# B&R Automation Studio project BottlePlant2
Automation Studio 4.10.2.37; technology packages: Acp10Arnc0 5.12.2, mapp 5.12.1, mappSafety 5.12.2

## Configuration Config1

CPU 4PPC70.0702-20W, AutomationRuntime B4.91, Build 4.1.2, Safety 0.0, Vc V4.72.3

### Task classes (Cpu.sw)
```
Cyclic#1 (cycle 2000 us):
  AxisCtrl <- Software.Code.AxisCtrl.prg
  RobVis <- Source.Misc.RobVis.prg
  MachineSta <- Software.Code.MachineCtrl.prg
DataObjects: Acp10sys
NcDataObjects: acp10etxen <- acp10etxen.dob, gTranAxisa <- gTranAxisobj.gTranAxisa.dob, gTranAxisi <- gTranAxisobj.gTranAxisi.dob, gCartAxisa <- gCartAxisobj.gCartAxisa.dob, gCartAxisi <- gCartAxisobj.gCartAxisi.dob, gPourAxisa <- gPourAxisobj.gPourAxisa.dob, gPourAxisi <- gPourAxisobj.gPourAxisi.dob
VcDataObjects: Visu <- Software.HMI.Visu.dob
Binaries: udbdef, arflatprv, TCData, arsvcreg, FWRules, arcoal, acp10cfg, Acp10map, sysconf, iomap, asfw, Transport, Role, ashwac, Cart, Pourer, arconfig, ashwd, User
Libraries: SfDomain, Acp10man, Acp10par, NcGlobal, Acp10sim, Acp10_MC, sys_lib, brsystem, runtime, MpAxis, MpBase, MpCom, astcp, asieccon, fileio, asbrstr, asiodiag, SfDomVis, astime, dataobj, SfDomDrv, asusb, MpSfDomMgr, aruser, powerlnk, standard, AsBrMath
```

### Task classes (AppMo.sw)
```

```

### Hardware
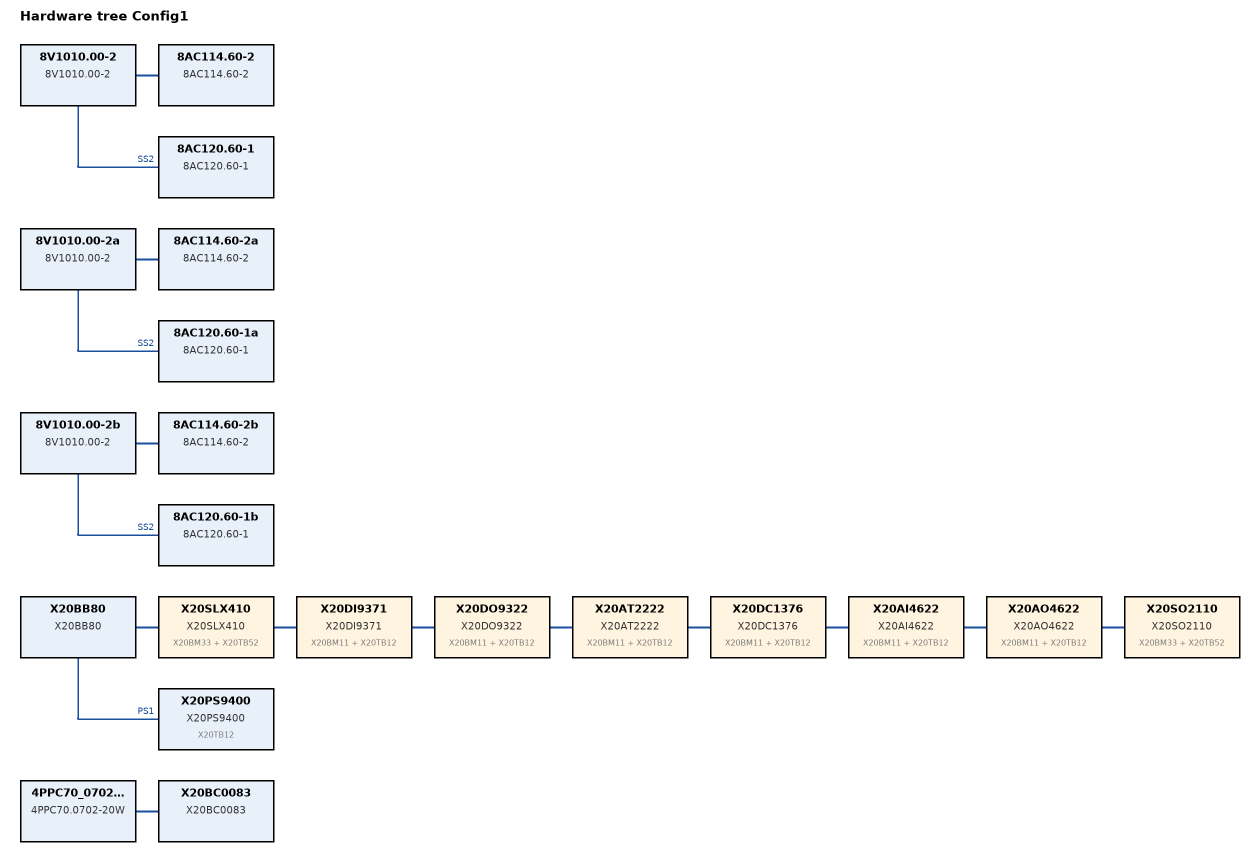
```
4PPC70_0702_20W : 4PPC70.0702-20W v1.5.2.0
  Connector IF2:
    ActivateDevice = 1
    Mode = Manual
    InternetAddress = 10.48.30.236
    SubnetMask = 255.255.255.0
    Vnc1
    VncVcObjectName1 = Visu
    VncKeyMappingFile1 = VC\PS2-Keyboard.dis
    VncRefreshRate1 = 100
    ActivateSnmp = 2
  ConfigurationID = BottlePlant2_Config1
  Simulation = 1
  TimerDeviceType = EPLX2X
  TimerDevice = 4PPC70_0702_20W.IF1
  TaskClassIdleTime = 2000
  Cyclic1Duration = 2000
  FileDevice1
  FileDeviceName1 = RecipeFile
  FileDevicePath1 = F:\Recipe
  FtpUser1
  FtpUsername1 = Admin
  FtpUserPassword1 = uT8p0uNS80JC7A4YbQtDpgpyP3aiMc7PVyx0K6ICeRY=
  FtpUserSalt1 = sviO6ryF
  FTPAccessRight1 = 0
  ActivateOpcUa = 1
  OpcUaInformationModels_PV_Version = 1
  VcObjectName = Visu
  KeyMappingFile = VC\4PPC70_0702_20W.dis
8AC114.60-2 : 8AC114.60-2 v1.0.0.8  [SS -> 8V1010.00-2.SS1; PLK1 -> X20BC0083.PLK2 (NodeNumber=4) [Cable Type=PowerlinkCable, Length=10, Version=1.0.0.3]; PLK2 -> 8AC114.60-2a.PLK1 (NodeNumber=4) [Cable Type=PowerlinkCable, Length=10, Version=1.0.0.3]]
8AC114.60-2a : 8AC114.60-2 v1.0.0.8  [SS -> 8V1010.00-2a.SS1; PLK1 -> 8AC114.60-2.PLK2 (NodeNumber=6) [Cable Type=PowerlinkCable, Length=10, Version=1.0.0.3]; PLK2 -> 8AC114.60-2b.PLK1 (NodeNumber=6) [Cable Type=PowerlinkCable, Length=10, Version=1.0.0.3]]
8AC114.60-2b : 8AC114.60-2 v1.0.0.8  [SS -> 8V1010.00-2b.SS1; PLK1 -> 8AC114.60-2a.PLK2 (NodeNumber=9) [Cable Type=PowerlinkCable, Length=10, Version=1.0.0.3]]
8AC120.60-1 : 8AC120.60-1 v2.2.0.0  [SS -> 8V1010.00-2.SS2]
8AC120.60-1a : 8AC120.60-1 v2.2.0.0  [SS -> 8V1010.00-2a.SS2]
8AC120.60-1b : 8AC120.60-1 v2.2.0.0  [SS -> 8V1010.00-2b.SS2]
8V1010.00-2 : 8V1010.00-2 v2.2.0.0
  MotionTP = Acp10Arnc0
  Simulate = standard
  PoweredBy = DC
  ActiveMotorSimulation_r1 = on
  BothEndSwitchesAreNormallyOpen_r1 = on
  QuickStopIsNormallyOpen_r1 = on
8V1010.00-2a : 8V1010.00-2 v2.2.0.0
  MotionTP = Acp10Arnc0
  Simulate = standard
  PoweredBy = DC
  ActiveMotorSimulation_r1 = on
  BothEndSwitchesAreNormallyOpen_r1 = on
  QuickStopIsNormallyOpen_r1 = on
8V1010.00-2b : 8V1010.00-2 v2.2.0.0
  MotionTP = Acp10Arnc0
  Simulate = standard
  PoweredBy = DC
  ActiveMotorSimulation_r1 = on
  BothEndSwitchesAreNormallyOpen_r1 = on
  QuickStopIsNormallyOpen_r1 = on
X20AI4622 : X20AI4622 v1.1.0.0  [SS1 -> X20TB12e.SS; SL -> X20BM11d.SL1]
  Supervision = off
X20AO4622 : X20AO4622 v1.2.0.0  [SS1 -> X20TB12f.SS; SL -> X20BM11e.SL1]
  Supervision = off
X20AT2222 : X20AT2222 v1.3.0.0  [SS1 -> X20TB12c.SS; SL -> X20BM11b.SL1]
  Supervision = off
X20BB80 : X20BB80 v1.0.2.0
X20BC0083 : X20BC0083 v2.11.1.0  [PLK1 -> 4PPC70_0702_20W.IF1 (NodeNumber=2) [Cable Type=PowerlinkCable, Length=10, Version=1.0.0.3]; PLK2 -> 8AC114.60-2.PLK1 (NodeNumber=2) [Cable Type=PowerlinkCable, Length=10, Version=1.0.0.3]; SL -> X20BB80.SL1]
  Supervision = off
X20BM11 : X20BM11 v1.0.0.1  [X2X1 -> X20BM33.X2X2]
X20BM11a : X20BM11 v1.0.0.1  [X2X1 -> X20BM11.X2X2]
X20BM11b : X20BM11 v1.0.0.1  [X2X1 -> X20BM11a.X2X2]
X20BM11c : X20BM11 v1.0.0.1  [X2X1 -> X20BM11b.X2X2]
X20BM11d : X20BM11 v1.0.0.1  [X2X1 -> X20BM11c.X2X2]
X20BM11e : X20BM11 v1.0.0.1  [X2X1 -> X20BM11d.X2X2]
X20BM33 : X20BM33 v1.0.0.6  [X2X1 -> X20BB80.IF1]
X20BM33a : X20BM33 v1.0.0.6  [X2X1 -> X20BM11e.X2X2]
X20DC1376 : X20DC1376 v1.2.0.0  [SS1 -> X20TB12d.SS; SL -> X20BM11c.SL1]
  Supervision = off
X20DI9371 : X20DI9371 v1.1.0.0  [SS1 -> X20TB12a.SS; SL -> X20BM11.SL1]
  Supervision = off
X20DO9322 : X20DO9322 v1.3.0.0  [SS1 -> X20TB12b.SS; SL -> X20BM11a.SL1]
  Supervision = off
X20PS9400 : X20PS9400 v1.5.0.0  [SS1 -> X20TB12.SS; PS -> X20BB80.PS1]
  Supervision = off
X20SLX410 : X20SLX410 v2.4.0.1  [SS1 -> X20TB52.SS; SL -> X20BM33.SL1]
  Supervision = off
X20SO2110 : X20SO2110 v2.2.1.0  [SS1 -> X20TB52a.SS; SL -> X20BM33a.SL1]
  Supervision = off
X20TB12 : X20TB12 v1.0.0.0
X20TB12a : X20TB12 v1.0.0.0
X20TB12b : X20TB12 v1.0.0.0
X20TB12c : X20TB12 v1.0.0.0
X20TB12d : X20TB12 v1.0.0.0
X20TB12e : X20TB12 v1.0.0.0
X20TB12f : X20TB12 v1.0.0.0
X20TB52 : X20TB52 v1.0.0.2
X20TB52a : X20TB52 v1.0.0.2
```

### IoMap.iom - 4PPC70_0702_20W/IoMap.iom
```iecst
VAR_CONFIG
	::SequencerC:DoPourer AT %QX."X20DO9322".DigitalOutput01;
END_VAR
```

### Acp10cfg.ncc - 4PPC70_0702_20W/Motion/Acp10cfg.ncc
```
NcConfiguration (Version=5.12.2, NcSwId=Acp10)
  ACP10CF1_typ:
    cnt_nettrc_rec_drive = 1500
    bufsize_trace_upload = 1200
    tc_nc_man_task = Cyclic #1
    glob_pv_as_ncobject = Yes
    ncsys_dl_broadcast = Yes
    ncsys_dl_acp_reset = Yes
    safemc_log_err_to_ax = Yes
    network_init:
      ncsw_init_execute = Yes
      automatic_execute = No
      node_nr_warning = Yes
      net_err_before_ncact = Yes
    nettrc:
      enter_parsecrec = Yes
      enter_ncaction = Yes
      save_ring_startidx = Yes
    cam_prof_download:
      cam_dat_dl_parallel = No
      tc_cam_dl_parallel = Task class for NC Manager task
    plk_if[0]:
      if_name = IF1
      tc_CycDat_PLCopen = Task class for NC Manager task
      mc_broadcast_extdat = No
```

### Acp10map.ncm - 4PPC70_0702_20W/Motion/Acp10map.ncm
```
NcMapping (NcSwId=Acp10, DisabledNodesAreHidden=False)
  NcObject gTranAxis (ModuleId=8V1010.00-2, Type=ncAXIS, Channel=1, AcoposSimulation=Standard, InitParameter=gTranAxisi, AcoposParameter=gTranAxisa, Disabled=FALSE, ModuleDisabled=FALSE)
  NcObject 8V1010.00-2_ncV_AXIS1 (ModuleId=8V1010.00-2, Type=ncV_AXIS, Channel=1, Disabled=TRUE, ModuleDisabled=FALSE)
  NcObject gCartAxis (ModuleId=8V1010.00-2a, Type=ncAXIS, Channel=1, AcoposSimulation=Standard, InitParameter=gCartAxisi, AcoposParameter=gCartAxisa, Disabled=FALSE, ModuleDisabled=FALSE)
  NcObject 8V1010.00-2a_ncV_AXIS1 (ModuleId=8V1010.00-2a, Type=ncV_AXIS, Channel=1, Disabled=TRUE, ModuleDisabled=FALSE)
  NcObject gPourAxis (ModuleId=8V1010.00-2b, Type=ncAXIS, Channel=1, AcoposSimulation=Standard, InitParameter=gPourAxisi, AcoposParameter=gPourAxisa, Disabled=FALSE, ModuleDisabled=FALSE)
  NcObject 8V1010.00-2b_ncV_AXIS1 (ModuleId=8V1010.00-2b, Type=ncV_AXIS, Channel=1, Disabled=TRUE, ModuleDisabled=FALSE)
```

### Cart.mpaxisbasic - 4PPC70_0702_20W/Motion/Config/Cart.mpaxisbasic
```
Element gCartAxisCfg (Type=mpaxisbasic)
  AxisConfiguration = AxisWithConfiguration
    Axis:
      BaseType = 4
    Drive:
      Controller:
        LoopFilters:
          [0]
          [1]
          [2]
Element gCartAxisCfg_1 (Type=mpaxisbasic)
```

### Pourer.mpaxisbasic - 4PPC70_0702_20W/Motion/Config/Pourer.mpaxisbasic
```
Element gPourAxisCfg (Type=mpaxisbasic)
  AxisConfiguration = AxisWithConfiguration
    Axis:
      BaseType = 4
      PeriodSettings:
        Period = 360
      MovementLimits:
        VelocityPositive = 1000
        VelocityNegative = 1000
        Acceleration = 5000
        Deceleration = 5000
    Drive:
      Controller:
        LoopFilters:
          [0]
          [1]
          [2]
```

### Transport.mpaxisbasic - 4PPC70_0702_20W/Motion/Config/Transport.mpaxisbasic
```
Element gTranAxisCfg (Type=mpaxisbasic)
  AxisConfiguration = AxisWithConfiguration
    Axis:
      BaseType = 4
      PeriodSettings:
        Period = 360
    Drive:
      Controller:
        LoopFilters:
          [0]
          [1]
          [2]
```

### Alarm.mpalarmbasic - 4PPC70_0702_20W/mappServices/Alarm/Alarm.mpalarmbasic
```
Element gAlarmBasic (Type=mpalarmbasic)
  mapp.Alarm.Factory:
    Reactions:
      Reaction[0]:
        Description = Example: Immediate Stop
  Alarms:
    UserAlarm:
      Alarms:
        Alarm[0]:
          Description = Example: Temperature over Tolerance
          Reaction = 1
```

### UserManagm.mpuser - 4PPC70_0702_20W/mappServices/User/UserManagm.mpuser
```
Element UserMgmt (Type=mpuser)
  Groups:
    DefGroup#1:
      id = Admin
      level = 100
      admin = TRUE
      rights:
        [0] = FullAccess
        [1] = FullAccess
        [2] = FullAccess
        [3] = FullAccess
        [4] = FullAccess
    DefGroup#2:
      id = Operator
      rights:
        [0] = FullAccess
        [1] = StartOnly
        [2] = ViewOnly
        [3] = ViewOnly
        [4] = NoAccess
    DefGroup#3:
      id = Supervisor
      level = 21
  Users:
    DefUser#1:
      id = Admin
      grp = Admin
      name = Default Admin User
      pwd = Admin
      pref = /LANG=0 /UNIT=0
    DefUser#2:
      id = macko
      grp = Operator
      pwd = 12345
    DefUser#3:
      id = supervisor1
      grp = Supervisor
      pwd = 12345
```

### UserSign.mpusersign - 4PPC70_0702_20W/mappServices/User/UserSign.mpusersign
```
Element gUserSign (Type=mpusersign)
```

## Logical view

Binary libraries used (declarations not repeated): operator, runtime, astime, AsIecCon, SfDomain 5.12.2, Acp10man, Acp10par, NcGlobal, Acp10sim, Acp10_MC, sys_lib, brsystem, MpAxis, MpBase, MpCom, standard, AsBrMath, MpRecipe, asstring, FileIO, MpUser 5.12.1, MpFile, MpAlarm 5.12.1

### Global.typ - Global data types
```iecst
(* AutoAxis *)
TYPE
	gAxesCtrlType : 	STRUCT
		Ctrl : gAxisBasicCtrlType;
		Cmd : gCmdType;
		State : gAutoAxisStateType;
		Timers : gTimersType;
		TimersPar : gTimersParType;
	END_STRUCT;
	gAxisBasicCtrlType : 	STRUCT
		MpTransporterAxis : MpAxisBasic;
		MpTransporterAxisPar : MpAxisBasicParType;
		MpCartAxis : MpAxisBasic;
		MpCartAxisPar : MpAxisBasicParType;
		MpPourerAxis : MpAxisBasic;
		MpPourerAxisPar : MpAxisBasicParType;
	END_STRUCT;
	gCmdType : 	STRUCT
		Power : BOOL;
		Home : BOOL;
		Update : BOOL;
		Stop : BOOL;
		ErrorReset : BOOL;
		MoveVelocity : BOOL;
		MoveAdditive : BOOL;
		MoveAbsolute : BOOL;
	END_STRUCT;

	gTimersType : STRUCT
		PowerTimer : ARRAY[0..2] OF TON;
		HomeTimer : ARRAY[0..2] OF TON;
	END_STRUCT;

	gTimersParType : STRUCT
		PowerDelayTime : REAL :=5;
		HomeDelayTime : REAL :=5;
	END_STRUCT;

	gAutoAxisStateType :
		(
		STATE_INIT_AXES := 0,
		STATE_WAIT_FOR_CMD_AXES := 1,
		STATE_POWER_ON_AXES := 2,
		STATE_HOME_AXES := 3,
		STATE_UPDATE_AXES := 4,
		STATE_MOVE_VELOCITY_AXES := 5,
		STATE_MOVE_ABSOLUTE_AXES := 6,
		STATE_MOVE_ADDITIVE_AXES := 7,
		STATE_STOP_AXES := 8,
		STATE_ERROR_AXES := 10
	);
END_TYPE
```

### Global.var - Global variables
```iecst
VAR
	gTranAxis : ACP10AXIS_typ;
	gCartAxis : ACP10AXIS_typ;
	gPourAxis : ACP10AXIS_typ;
END_VAR
```


### Program Logical/Software/Code/AxisCtrl (IEC)

#### Main.st
```iecst
PROGRAM _INIT
	(* Insert code here *)
	gAxes.SequencerCtrl.MpAxisCamSequencer_0.Enable:=TRUE;
	gAxes.SequencerCtrl.MpAxisCamSequencer_1.Enable:=TRUE;

	gAxes.SequencerCtrl.MpAxisCamSequencerPar_0.Deceleration:=1000;
	gAxes.SequencerCtrl.MpAxisCamSequencerPar_0.Configuration.Master:=ADR(gTranAxis);
	gAxes.SequencerCtrl.MpAxisCamSequencerPar_0.Configuration.StartState:=0;
	gAxes.SequencerCtrl.MpAxisCamSequencerPar_0.Configuration.State[0].Event[0].Type:=ncS_START;
	gAxes.SequencerCtrl.MpAxisCamSequencerPar_0.Configuration.State[0].Event[0].Attribute:=ncAT_ONCE;
	gAxes.SequencerCtrl.MpAxisCamSequencerPar_0.Configuration.State[0].Event[0].NextState:=1;

	gAxes.SequencerCtrl.MpAxisCamSequencerPar_0.Configuration.State[1].CompMode:=ncONLYCOMP_DIRECT;
	gAxes.SequencerCtrl.MpAxisCamSequencerPar_0.Configuration.State[1].CamProfileIndex:=16#ffff;

	gAxes.SequencerCtrl.MpAxisCamSequencerPar_0.Configuration.State[1].MasterCompDistance:=0;
	gAxes.SequencerCtrl.MpAxisCamSequencerPar_0.Configuration.State[1].SlaveCompDistance:=0;

	gAxes.SequencerCtrl.MpAxisCamSequencerPar_0.Configuration.State[1].MasterFactor:=400*100;
	gAxes.SequencerCtrl.MpAxisCamSequencerPar_0.Configuration.State[1].SlaveFactor:=400*100;

	gAxes.SequencerCtrl.MpAxisCamSequencerPar_0.Configuration.State[1].Event[0].Type:=ncST_END;
	gAxes.SequencerCtrl.MpAxisCamSequencerPar_0.Configuration.State[1].Event[0].Attribute:=ncAT_ONCE;
	gAxes.SequencerCtrl.MpAxisCamSequencerPar_0.Configuration.State[1].Event[0].NextState:=2;

	gAxes.SequencerCtrl.MpAxisCamSequencerPar_0.Configuration.State[2].CompMode:=ncONLYCOMP_DIRECT;
	gAxes.SequencerCtrl.MpAxisCamSequencerPar_0.Configuration.State[2].CamProfileIndex:=16#fffe;

	gAxes.SequencerCtrl.MpAxisCamSequencerPar_0.Configuration.State[2].MasterCompDistance:=100;
	gAxes.SequencerCtrl.MpAxisCamSequencerPar_0.Configuration.State[2].SlaveCompDistance:=-400;

	gAxes.SequencerCtrl.MpAxisCamSequencerPar_0.Configuration.State[2].MasterFactor:=1;
	gAxes.SequencerCtrl.MpAxisCamSequencerPar_0.Configuration.State[2].SlaveFactor:=1;

	gAxes.SequencerCtrl.MpAxisCamSequencerPar_0.Configuration.State[2].Event[0].Type:=ncST_END;
	gAxes.SequencerCtrl.MpAxisCamSequencerPar_0.Configuration.State[2].Event[0].Attribute:=ncAT_ONCE;
	gAxes.SequencerCtrl.MpAxisCamSequencerPar_0.Configuration.State[2].Event[0].NextState:=1;

	(* drugi seq *)

	gAxes.SequencerCtrl.MpAxisCamSequencerPar_1.Deceleration:=1000;
	gAxes.SequencerCtrl.MpAxisCamSequencerPar_1.Configuration.Master:=ADR(gCartAxis);
	gAxes.SequencerCtrl.MpAxisCamSequencerPar_1.Configuration.StartState:=0;
	gAxes.SequencerCtrl.MpAxisCamSequencerPar_1.Configuration.State[0].Event[0].Type:=ncSIGNAL1;
	gAxes.SequencerCtrl.MpAxisCamSequencerPar_1.Configuration.State[0].Event[0].Attribute:=ncAT_ONCE;
	gAxes.SequencerCtrl.MpAxisCamSequencerPar_1.Configuration.State[0].Event[0].NextState:=1;

	gAxes.SequencerCtrl.MpAxisCamSequencerPar_1.Configuration.State[1].CompMode:=ncONLYCOMP_DIRECT;
	gAxes.SequencerCtrl.MpAxisCamSequencerPar_1.Configuration.State[1].CamProfileIndex:=16#fffe;
	gAxes.SequencerCtrl.MpAxisCamSequencerPar_1.Configuration.State[1].MasterCompDistance:=100.0;
	gAxes.SequencerCtrl.MpAxisCamSequencerPar_1.Configuration.State[1].SlaveCompDistance:=275.0;
	gAxes.SequencerCtrl.MpAxisCamSequencerPar_1.Configuration.State[1].MasterFactor:=1;
	gAxes.SequencerCtrl.MpAxisCamSequencerPar_1.Configuration.State[1].SlaveFactor:=0;
	gAxes.SequencerCtrl.MpAxisCamSequencerPar_1.Configuration.State[1].Event[0].Type:=ncST_END;
	gAxes.SequencerCtrl.MpAxisCamSequencerPar_1.Configuration.State[1].Event[0].Attribute:=ncAT_ONCE;
	gAxes.SequencerCtrl.MpAxisCamSequencerPar_1.Configuration.State[1].Event[0].NextState:=2;

	//	gAxes.SequencerCtrl.MpAxisCamSequencerPar_1.Configuration.State[2].CompMode:=ncONLYCOMP_DIRECT;
	//	gAxes.SequencerCtrl.MpAxisCamSequencerPar_1.Configuration.State[2].CamProfileIndex:=16#ffff;
	//	gAxes.SequencerCtrl.MpAxisCamSequencerPar_1.Configuration.State[2].MasterCompDistance:=0.0;
	//	gAxes.SequencerCtrl.MpAxisCamSequencerPar_1.Configuration.State[2].SlaveCompDistance:=0.0;
	//	gAxes.SequencerCtrl.MpAxisCamSequencerPar_1.Configuration.State[2].MasterFactor:=200*100;
	//	gAxes.SequencerCtrl.MpAxisCamSequencerPar_1.Configuration.State[2].SlaveFactor:=0;
	//	gAxes.SequencerCtrl.MpAxisCamSequencerPar_1.Configuration.State[2].Event[0].Type:=ncST_END;
	//	gAxes.SequencerCtrl.MpAxisCamSequencerPar_1.Configuration.State[2].Event[0].Attribute:=ncAT_ONCE;
	//	gAxes.SequencerCtrl.MpAxisCamSequencerPar_1.Configuration.State[2].Event[0].NextState:=3;

	gAxes.SequencerCtrl.MpAxisCamSequencerPar_1.Configuration.State[2].CompMode:=ncONLYCOMP_DIRECT;
	gAxes.SequencerCtrl.MpAxisCamSequencerPar_1.Configuration.State[2].CamProfileIndex:=16#fffe;
	gAxes.SequencerCtrl.MpAxisCamSequencerPar_1.Configuration.State[2].MasterCompDistance:=290.0;
	gAxes.SequencerCtrl.MpAxisCamSequencerPar_1.Configuration.State[2].SlaveCompDistance:=-275.0;
	gAxes.SequencerCtrl.MpAxisCamSequencerPar_1.Configuration.State[2].MasterFactor:=1;
	gAxes.SequencerCtrl.MpAxisCamSequencerPar_1.Configuration.State[2].SlaveFactor:=0;
	gAxes.SequencerCtrl.MpAxisCamSequencerPar_1.Configuration.State[2].Event[0].Type:=ncST_END;
	gAxes.SequencerCtrl.MpAxisCamSequencerPar_1.Configuration.State[2].Event[0].Attribute:=ncAT_ONCE;
	gAxes.SequencerCtrl.MpAxisCamSequencerPar_1.Configuration.State[2].Event[0].NextState:=0;

	gAxes.SequencerCtrl.MpAxisCamSequencerPar_1.Configuration.State[3].CompMode:=ncONLYCOMP_DIRECT;
	gAxes.SequencerCtrl.MpAxisCamSequencerPar_1.Configuration.State[3].CamProfileIndex:=16#fffe;
	gAxes.SequencerCtrl.MpAxisCamSequencerPar_1.Configuration.State[3].MasterCompDistance:=90.0;
	gAxes.SequencerCtrl.MpAxisCamSequencerPar_1.Configuration.State[3].SlaveCompDistance:=-470.0;
	gAxes.SequencerCtrl.MpAxisCamSequencerPar_1.Configuration.State[3].MasterFactor:=1;
	gAxes.SequencerCtrl.MpAxisCamSequencerPar_1.Configuration.State[3].SlaveFactor:=0;
	gAxes.SequencerCtrl.MpAxisCamSequencerPar_1.Configuration.State[3].Event[0].Type:=ncST_END;
	gAxes.SequencerCtrl.MpAxisCamSequencerPar_1.Configuration.State[3].Event[0].Attribute:=ncAT_ONCE;
	gAxes.SequencerCtrl.MpAxisCamSequencerPar_1.Configuration.State[3].Event[0].NextState:=0;
	(* To DO -> timer w homming, brak wylaczania zasilani *)
	gAxes.State.Auto:=STATE_INIT_AXES;
	gControlType:=TRUE;
END_PROGRAM

PROGRAM _CYCLIC
	(* Insert code here *)
	gAxes.Ctrl.MpTransporterAxis.MpLink:=ADR(gTranAxisCfg);
	gAxes.Ctrl.MpTransporterAxis.Parameters:=ADR(gAxes.Ctrl.MpTransporterAxisPar);
	gAxes.Ctrl.MpTransporterAxis.Axis:=ADR(gTranAxis);

	gAxes.Ctrl.MpCartAxis.MpLink:=ADR(gCartAxisCfg);
	gAxes.Ctrl.MpCartAxis.Parameters:=ADR(gAxes.Ctrl.MpCartAxisPar);
	gAxes.Ctrl.MpCartAxis.Axis:=ADR(gCartAxis);

	gAxes.Ctrl.MpPourerAxis.MpLink:=ADR(gPourAxisCfg);
	gAxes.Ctrl.MpPourerAxis.Parameters:=ADR(gAxes.Ctrl.MpPourerAxisPar);
	gAxes.Ctrl.MpPourerAxis.Axis:=ADR(gPourAxis);

	gAxes.SequencerCtrl.MpAxisCamSequencer_0.MpLink:=ADR(gCartAxisCfg);
	gAxes.SequencerCtrl.MpAxisCamSequencer_0.MpLinkMaster:=ADR(gTranAxisCfg);
	gAxes.SequencerCtrl.MpAxisCamSequencer_0.Parameters:=ADR(gAxes.SequencerCtrl.MpAxisCamSequencerPar_0);
	gAxes.SequencerCtrl.MpAxisCamSequencer_0();

	gAxes.SequencerCtrl.MpAxisCamSequencer_1.MpLink:=ADR(gPourAxisCfg);
	gAxes.SequencerCtrl.MpAxisCamSequencer_1.MpLinkMaster:=ADR(gCartAxisCfg);
	gAxes.SequencerCtrl.MpAxisCamSequencer_1.Parameters:=ADR(gAxes.SequencerCtrl.MpAxisCamSequencerPar_1);
	//Machine.SequencerCtrl.MpAxisCamSequencer_1.Signal1:=Machine.SequencerCtrl.MpAxisCamSequencer_0.InCompensation;
	gAxes.SequencerCtrl.MpAxisCamSequencer_1();

	gAxes.Ctrl.MpTransporterAxis();
	gAxes.Ctrl.MpCartAxis();
	gAxes.Ctrl.MpPourerAxis();

	(* MAszyna stanów zarządzajaca silnikami *)
	IF gAxes.Ctrl.MpTransporterAxis.Error THEN
		//alarm osi transporter
		gAxes.State.Auto:=STATE_ERROR_AXES;
	END_IF
	IF gAxes.Ctrl.MpCartAxis.Error THEN
		//alarm osi wozka
		gAxes.State.Auto:=STATE_ERROR_AXES;
	END_IF
	IF gAxes.Ctrl.MpPourerAxis.Error THEN
		//alarm nalewaka
		gAxes.State.Auto:=STATE_ERROR_AXES;
	END_IF

	CASE gAxes.State.Auto OF
		STATE_INIT_AXES:
			gAxes.Ctrl.MpTransporterAxis.Enable:=TRUE;
			gAxes.Ctrl.MpCartAxis.Enable:=TRUE;
			gAxes.Ctrl.MpPourerAxis.Enable:=TRUE;

			IF gAxes.Ctrl.MpTransporterAxis.Active AND gAxes.Ctrl.MpCartAxis.Active AND gAxes.Ctrl.MpPourerAxis.Active THEN
				gAxes.State.Auto:=STATE_POWER_ON_AXES;
			END_IF;
		STATE_WAIT_FOR_CMD_AXES:
			IF EDGEPOS(gAxes.Cmd.Auto.Power) THEN
				gAxes.Cmd.Auto.Power:=FALSE;
				gAxes.State.Auto:=STATE_POWER_ON_AXES;
			ELSIF EDGEPOS(gAxes.Cmd.Auto.Home) THEN
				gAxes.Cmd.Auto.Home:=FALSE;
				gAxes.State.Auto:=STATE_HOME_AXES;
			ELSIF EDGEPOS(gAxes.Cmd.Auto.Update) THEN
				gAxes.Cmd.Auto.Update:=FALSE;
				gAxes.State.Auto:=STATE_UPDATE_AXES;
			ELSIF EDGEPOS(gAxes.Cmd.Auto.Stop) THEN
				gAxes.Cmd.Auto.Stop:=FALSE;
				gAxes.State.Auto:=STATE_STOP_AXES;
			ELSIF EDGEPOS(gAxes.Cmd.Auto.ErrorReset) THEN
				gAxes.Cmd.Auto.ErrorReset:=FALSE;
			ELSIF EDGEPOS(gAxes.Cmd.Auto.MoveVelocity) THEN
				gAxes.Cmd.Auto.MoveVelocity:=FALSE;
				gAxes.State.Auto:=STATE_MOVE_VELOCITY_AXES;
//				ELSIF gAxes.Cmd.Auto.MoveAbsolute THEN
//				ELSIF gAxes.Cmd.Auto.MoveAdditive THEN
			END_IF;
		STATE_POWER_ON_AXES:
			gAxes.Ctrl.MpTransporterAxis.Power:=TRUE;
			gAxes.Ctrl.MpCartAxis.Power:=TRUE;
			gAxes.Ctrl.MpPourerAxis.Power:=TRUE;

			gAxes.Timers.PowerTimer[0].IN:=NOT(gAxes.Ctrl.MpTransporterAxis.PowerOn);
			gAxes.Timers.PowerTimer[0].PT:=REAL_TO_TIME(gAxes.TimersPar.PowerDelayTime*1000);
			gAxes.Timers.PowerTimer[0]();

			gAxes.Timers.PowerTimer[1].IN:=NOT(gAxes.Ctrl.MpCartAxis.PowerOn);
			gAxes.Timers.PowerTimer[1].PT:=REAL_TO_TIME(gAxes.TimersPar.PowerDelayTime*1000);
			gAxes.Timers.PowerTimer[1]();

			gAxes.Timers.PowerTimer[2].IN:=NOT(gAxes.Ctrl.MpPourerAxis.PowerOn);
			gAxes.Timers.PowerTimer[2].PT:=REAL_TO_TIME(gAxes.TimersPar.PowerDelayTime*1000);
			gAxes.Timers.PowerTimer[2]();

			IF gAxes.Timers.PowerTimer[0].Q THEN
				//zbyt dlugie zalaczanie osi transportra alarm
				gAxes.Timers.PowerTimer[0].IN:=FALSE;
				gAxes.Timers.PowerTimer[0]();
				gAxes.State.Auto:=STATE_ERROR_AXES;
			END_IF;
			IF gAxes.Timers.PowerTimer[1].Q THEN
				//zbyt dlugie zalaczanie osi wozka alarm
				gAxes.Timers.PowerTimer[1].IN:=FALSE;
				gAxes.Timers.PowerTimer[1]();
				gAxes.State.Auto:=STATE_ERROR_AXES;
			END_IF;
			IF gAxes.Timers.PowerTimer[2].Q THEN
				//zbyt dlugie zalaczanie osi nalewaka alarm
				gAxes.Timers.PowerTimer[2].IN:=FALSE;
				gAxes.Timers.PowerTimer[2]();
				gAxes.State.Auto:=STATE_ERROR_AXES;
			END_IF;

			IF gAxes.Ctrl.MpTransporterAxis.PowerOn AND gAxes.Ctrl.MpCartAxis.PowerOn AND gAxes.Ctrl.MpPourerAxis.PowerOn THEN
				gAxes.State.Auto:=STATE_WAIT_FOR_CMD_AXES;
				gAxes.Timers.PowerTimer[0].IN:=FALSE;
				gAxes.Timers.PowerTimer[0]();
				gAxes.Timers.PowerTimer[1].IN:=FALSE;
				gAxes.Timers.PowerTimer[1]();
				gAxes.Timers.PowerTimer[2].IN:=FALSE;
				gAxes.Timers.PowerTimer[2]();
			END_IF;

		STATE_HOME_AXES:
			gAxes.Ctrl.MpTransporterAxis.Home:=TRUE;
			gAxes.Ctrl.MpCartAxis.Home:=gAxes.Ctrl.MpTransporterAxis.IsHomed;
			gAxes.Ctrl.MpPourerAxis.Home:=gAxes.Ctrl.MpCartAxis.IsHomed;

			gAxes.Timers.HomeTimer[0].IN:=NOT(gAxes.Ctrl.MpTransporterAxis.IsHomed);
			gAxes.Timers.HomeTimer[0].PT:=REAL_TO_TIME(gAxes.TimersPar.HomeDelayTime*1000);
			gAxes.Timers.HomeTimer[0]();

			gAxes.Timers.HomeTimer[1].IN:=gAxes.Ctrl.MpTransporterAxis.IsHomed AND NOT(gAxes.Ctrl.MpCartAxis.IsHomed);
			gAxes.Timers.HomeTimer[1].PT:=REAL_TO_TIME(gAxes.TimersPar.HomeDelayTime*1000);
			gAxes.Timers.HomeTimer[1]();

			gAxes.Timers.HomeTimer[2].IN:=gAxes.Ctrl.MpCartAxis.IsHomed AND NOT(gAxes.Ctrl.MpPourerAxis.IsHomed);
			gAxes.Timers.HomeTimer[2].PT:=REAL_TO_TIME(gAxes.TimersPar.HomeDelayTime*1000);
			gAxes.Timers.HomeTimer[2]();

			IF gAxes.Timers.HomeTimer[0].Q THEN
				gAxes.Timers.HomeTimer[0].IN:=FALSE;
				gAxes.Timers.HomeTimer[0]();
				//zbyt dlugie bazowanie osi transportra alarm
				gAxes.State.Auto:=STATE_ERROR_AXES;
			END_IF;

			IF gAxes.Timers.HomeTimer[1].Q THEN
				gAxes.Timers.HomeTimer[1].IN:=FALSE;
				gAxes.Timers.HomeTimer[1]();
				//zbyt dlugie bazowanie osi wozka alarm
				gAxes.State.Auto:=STATE_ERROR_AXES;
			END_IF;

			IF gAxes.Timers.HomeTimer[2].Q THEN
				gAxes.Timers.HomeTimer[2].IN:=FALSE;
				gAxes.Timers.HomeTimer[2]();
				//zbyt dlugie bazowanie osi nalewaka alarm
				gAxes.State.Auto:=STATE_ERROR_AXES;
			END_IF;

			IF gAxes.Ctrl.MpTransporterAxis.IsHomed AND gAxes.Ctrl.MpCartAxis.IsHomed AND gAxes.Ctrl.MpPourerAxis.IsHomed THEN
				gAxes.Ctrl.MpTransporterAxis.Home:=FALSE;
				gAxes.Ctrl.MpCartAxis.Home:=FALSE;
				gAxes.Ctrl.MpPourerAxis.Home:=FALSE;
				gAxes.State.Auto:=STATE_WAIT_FOR_CMD_AXES;
				gAxes.Timers.HomeTimer[0].IN:=FALSE;
				gAxes.Timers.HomeTimer[0]();
				gAxes.Timers.HomeTimer[1].IN:=FALSE;
				gAxes.Timers.HomeTimer[1]();
				gAxes.Timers.HomeTimer[2].IN:=FALSE;
				gAxes.Timers.HomeTimer[2]();
			END_IF;
		STATE_STOP_AXES:
			//bez wylaczania zasialania
			(* Sprawdzenie czy jes wlaczonysilnik jesi tak to stop - jesli off to wywalierror *)
			IF gAxes.Ctrl.MpTransporterAxis.PowerOn THEN
				gAxes.Ctrl.MpTransporterAxis.Stop:=TRUE;
			END_IF;

			IF gAxes.Ctrl.MpCartAxis.PowerOn THEN
				gAxes.Ctrl.MpCartAxis.Stop:=TRUE;
			END_IF;

			IF gAxes.Ctrl.MpPourerAxis.PowerOn THEN
				gAxes.Ctrl.MpPourerAxis.Stop:=TRUE;
			END_IF;

			IF gAxes.Ctrl.MpTransporterAxis.Stopped AND gAxes.Ctrl.MpCartAxis.Stopped AND gAxes.Ctrl.MpPourerAxis.Stopped THEN
				gAxes.Ctrl.MpTransporterAxis.Stop:=FALSE;
				gAxes.Ctrl.MpCartAxis.Stop:=FALSE;
				gAxes.Ctrl.MpPourerAxis.Stop:=FALSE;
				gAxes.Ctrl.MpTransporterAxis.MoveVelocity:=FALSE;
				//gAxes.SequencerCtrl.MpAxisCamSequencer_0.StartSequence:=FALSE;
				//gAxes.SequencerCtrl.MpAxisCamSequencer_1.StartSequence:=FALSE;

				gAxes.State.Auto:=STATE_WAIT_FOR_CMD_AXES;
			END_IF;
		STATE_UPDATE_AXES:
			gAxes.Ctrl.MpTransporterAxis.Update:=TRUE;
			gAxes.Ctrl.MpCartAxis.Update:=TRUE;
			gAxes.Ctrl.MpPourerAxis.Update:=TRUE;

			IF gAxes.Ctrl.MpTransporterAxis.UpdateDone AND gAxes.Ctrl.MpCartAxis.UpdateDone AND gAxes.Ctrl.MpPourerAxis.UpdateDone THEN
				gAxes.State.Auto:=STATE_WAIT_FOR_CMD_AXES;
				gAxes.Ctrl.MpTransporterAxis.Update:=FALSE;
				gAxes.Ctrl.MpCartAxis.Update:=FALSE;
				gAxes.Ctrl.MpPourerAxis.Update:=FALSE;
			END_IF;
		STATE_MOVE_VELOCITY_AXES:
			(* Chyba że tu tdac ze ready  *)
			gAxes.SequencerCtrl.MpAxisCamSequencer_0.StartSequence:=TRUE;
			gAxes.SequencerCtrl.MpAxisCamSequencer_1.StartSequence:=TRUE;
			gAxes.Ctrl.MpTransporterAxis.MoveVelocity:=TRUE;
			gAxes.State.Auto:=STATE_WAIT_FOR_CMD_AXES;
		STATE_ERROR_AXES:
			(* Zatrzymanie wszystkich silnikow *)
			gAxes.Ctrl.MpTransporterAxis.MoveVelocity:=FALSE;
			IF gAxes.Ctrl.MpTransporterAxis.PowerOn THEN
				gAxes.Ctrl.MpTransporterAxis.Stop:=TRUE;
			END_IF;

			IF gAxes.Ctrl.MpCartAxis.PowerOn THEN
				gAxes.Ctrl.MpCartAxis.Stop:=TRUE;
			END_IF;

			IF gAxes.Ctrl.MpPourerAxis.PowerOn THEN
				gAxes.Ctrl.MpPourerAxis.Stop:=TRUE;
			END_IF;

			(* Jesli sa zastopowane to power off  *)
			IF gAxes.Ctrl.MpTransporterAxis.Stopped THEN
				gAxes.Ctrl.MpTransporterAxis.Power:=FALSE;
			END_IF;

			IF gAxes.Ctrl.MpCartAxis.Stopped THEN
				gAxes.Ctrl.MpCartAxis.Power:=FALSE;
			END_IF;

			IF gAxes.Ctrl.MpPourerAxis.Stopped THEN
				gAxes.Ctrl.MpPourerAxis.Power:=FALSE;
			END_IF;

			(* Czekamy na przycisk reseterror *)
			IF EDGEPOS(gAxes.Cmd.Auto.ErrorReset) AND (NOT(gAxes.Ctrl.MpTransporterAxis.PowerOn) AND NOT(gAxes.Ctrl.MpCartAxis.PowerOn) AND NOT(gAxes.Ctrl.MpPourerAxis.PowerOn)) THEN
				gAxes.Cmd.Auto.ErrorReset:=FALSE;

				gAxes.Ctrl.MpTransporterAxis.Stop:=FALSE;
				gAxes.Ctrl.MpCartAxis.Stop:=FALSE;
				gAxes.Ctrl.MpPourerAxis.Stop:=FALSE;

				gAxes.Ctrl.MpTransporterAxis.ErrorReset:=TRUE;
				gAxes.Ctrl.MpCartAxis.ErrorReset:=TRUE;
				gAxes.Ctrl.MpPourerAxis.ErrorReset:=TRUE;
				//gAxes.State.Auto:=WAIT_FOR_CMD;
			END_IF;

			IF NOT(gAxes.Ctrl.MpTransporterAxis.Error) AND NOT(gAxes.Ctrl.MpCartAxis.Error) AND NOT(gAxes.Ctrl.MpPourerAxis.Error) THEN
				gAxes.Ctrl.MpTransporterAxis.ErrorReset:=FALSE;
				gAxes.Ctrl.MpCartAxis.ErrorReset:=FALSE;
				gAxes.Ctrl.MpPourerAxis.ErrorReset:=FALSE;
				gAxes.State.Auto:=STATE_WAIT_FOR_CMD_AXES;
				//gAxes.Ctrl.MpTransporterAxis.MoveVelocity:=FALSE;
			END_IF
	END_CASE;

	CASE gAxes.State.Manual OF
		STATE_WAIT_FOR_CMD_MANUAL:
			gAxes.Ctrl.MpTransporterAxis.JogPositive:=gAxes.Cmd.Manual.TransporterJogPositive;
			gAxes.Ctrl.MpTransporterAxis.JogNegative:=gAxes.Cmd.Manual.TransporterJogNegative;

			gAxes.Ctrl.MpCartAxis.JogPositive:=gAxes.Cmd.Manual.CartJogPositive;
			gAxes.Ctrl.MpCartAxis.JogNegative:=gAxes.Cmd.Manual.CartJogNegative;

			gAxes.Ctrl.MpPourerAxis.JogPositive:=gAxes.Cmd.Manual.PourerJogPositive;
			gAxes.Ctrl.MpPourerAxis.JogNegative:=gAxes.Cmd.Manual.PourerJogNegative;

			IF EDGEPOS(gAxes.Cmd.Manual.TransporterHomming) THEN
				gAxes.Cmd.Manual.TransporterHomming:=FALSE;
				gAxes.State.Manual:=STATE_TRANSPORTER_HOMMING;
			ELSIF EDGEPOS(gAxes.Cmd.Manual.CartHomming)  THEN
				gAxes.Cmd.Manual.CartHomming:=FALSE;
				gAxes.State.Manual:=STATE_CART_HOMMING;
			ELSIF EDGEPOS(gAxes.Cmd.Manual.PourerHomming) THEN
				gAxes.Cmd.Manual.PourerHomming:=FALSE;
				gAxes.State.Manual:=STATE_POURER_HOMMING;
			END_IF;
		STATE_TRANSPORTER_HOMMING:
			gAxes.Ctrl.MpTransporterAxis.Home:=TRUE;
			gAxes.Timers.HomeTimer[0].IN:=NOT(gAxes.Ctrl.MpTransporterAxis.IsHomed);
			gAxes.Timers.HomeTimer[0].PT:=REAL_TO_TIME(gAxes.TimersPar.HomeDelayTime*1000);
			gAxes.Timers.HomeTimer[0]();

			IF gAxes.Timers.HomeTimer[0].Q THEN
				gAxes.Timers.HomeTimer[0].IN:=FALSE;
				gAxes.Timers.HomeTimer[0]();
				//zbyt dlugie bazowanie osi transportra alarm
				gAxes.State.Auto:=STATE_ERROR_AXES;
			END_IF;

			IF gAxes.Ctrl.MpTransporterAxis.IsHomed THEN
				gAxes.Ctrl.MpTransporterAxis.Home:=FALSE;
				gAxes.State.Manual:=STATE_WAIT_FOR_CMD_MANUAL;
				gAxes.Timers.HomeTimer[0].IN:=FALSE;
				gAxes.Timers.HomeTimer[0]();
			END_IF;
		STATE_CART_HOMMING:
			gAxes.Ctrl.MpCartAxis.Home:=TRUE;
			gAxes.Timers.HomeTimer[0].IN:=NOT(gAxes.Ctrl.MpCartAxis.IsHomed);
			gAxes.Timers.HomeTimer[0].PT:=REAL_TO_TIME(gAxes.TimersPar.HomeDelayTime*1000);
			gAxes.Timers.HomeTimer[0]();

			IF gAxes.Timers.HomeTimer[0].Q THEN
				gAxes.Timers.HomeTimer[0].IN:=FALSE;
				gAxes.Timers.HomeTimer[0]();
				//zbyt dlugie bazowanie osi MpCartAxis alarm
				gAxes.State.Auto:=STATE_ERROR_AXES;
			END_IF;

			IF gAxes.Ctrl.MpCartAxis.IsHomed THEN
				gAxes.Ctrl.MpCartAxis.Home:=FALSE;
				gAxes.State.Manual:=STATE_WAIT_FOR_CMD_MANUAL;
				gAxes.Timers.HomeTimer[0].IN:=FALSE;
				gAxes.Timers.HomeTimer[0]();
			END_IF;
		STATE_POURER_HOMMING:
			gAxes.Ctrl.MpPourerAxis.Home:=TRUE;
			gAxes.Timers.HomeTimer[0].IN:=NOT(gAxes.Ctrl.MpPourerAxis.IsHomed);
			gAxes.Timers.HomeTimer[0].PT:=REAL_TO_TIME(gAxes.TimersPar.HomeDelayTime*1000);
			gAxes.Timers.HomeTimer[0]();

			IF gAxes.Timers.HomeTimer[0].Q THEN
				gAxes.Timers.HomeTimer[0].IN:=FALSE;
				gAxes.Timers.HomeTimer[0]();
				//zbyt dlugie bazowanie osi MpCartAxis alarm
				gAxes.State.Auto:=STATE_ERROR_AXES;
			END_IF;

			IF gAxes.Ctrl.MpPourerAxis.IsHomed THEN
				gAxes.Ctrl.MpPourerAxis.Home:=FALSE;
				gAxes.State.Manual:=STATE_WAIT_FOR_CMD_MANUAL;
				gAxes.Timers.HomeTimer[0].IN:=FALSE;
				gAxes.Timers.HomeTimer[0]();
			END_IF;

	END_CASE;

	IF gAxes.SequencerCtrl.MpAxisCamSequencer_0.ActualStateIndex=1 THEN
		gAxes.SequencerCtrl.MpAxisCamSequencer_1.Signal1:=TRUE;
	ELSE
		gAxes.SequencerCtrl.MpAxisCamSequencer_1.Signal1:=FALSE;
	END_IF;
END_PROGRAM

PROGRAM _EXIT
	(* Insert code here *)
	gAxes.Ctrl.MpTransporterAxis.Power:=FALSE;
	gAxes.Ctrl.MpTransporterAxis.Enable:=FALSE;
	gAxes.Ctrl.MpTransporterAxis();

	gAxes.Ctrl.MpCartAxis.Power:=FALSE;
	gAxes.Ctrl.MpCartAxis.Enable:=FALSE;
	gAxes.Ctrl.MpCartAxis();

	gAxes.Ctrl.MpPourerAxis.Power:=FALSE;
	gAxes.Ctrl.MpPourerAxis.Enable:=FALSE;
	gAxes.Ctrl.MpPourerAxis();

END_PROGRAM
```

### Program Logical/Software/Code/MachineCtrl (IEC)

#### Types.typ
```iecst
TYPE
	MachineStateType :
		(
		STATE_INIT_MACHINE := 0,
		STATE_WAIT_FOR_CMD_MACHINE := 1,
		STATE_START_MACHINE:=2,
		STATE_STOP_MACHINE:=3,
		STATE_HOME_MACHINE := 4,
		STATE_MANUAL_MACHINE := 5,
		STATE_AUTO_MACHINE := 7,
		STATE_SERWIS_MACHINE := 8,
		STATE_ALARM_MACHINE := 9
	);
	StatesType : 	STRUCT
		MachineState : MachineStateType;
	END_STRUCT;

	CmdType : 	STRUCT
		MachineCmd : MachineCmdType;
	END_STRUCT;

	MachineCmdType : 	STRUCT
		Start : BOOL;
		Stop : BOOL;
		EStop : BOOL;
		Home : BOOL;
		AutoCtrl : BOOL;
		ManualCtrl : BOOL;
	END_STRUCT;

	GUIType : STRUCT
		uiShowLayer : ARRAY[0..5] OF INT;
	END_STRUCT;

	MachineCtrlType : 	STRUCT
		States : StatesType;
		Cmd : CmdType;
		GUI : GUIType;
	END_STRUCT;
END_TYPE
```

#### Variables.var
```iecst
VAR
	Machine :  MachineCtrlType;

END_VAR
```

#### Main.st
```iecst
PROGRAM _INIT
	(* Insert code here *)
	Machine.States.MachineState:=STATE_INIT_MACHINE;

END_PROGRAM

PROGRAM _CYCLIC
	(* Insert code here *)

	CASE Machine.States.MachineState OF
		STATE_INIT_MACHINE:
			IF gAxes.State.Auto=STATE_WAIT_FOR_CMD_AXES THEN
				Machine.GUI.uiShowLayer[0]:=0;
			END_IF;
			//jeden przycisk do home ktory pozwala zbazowac wszystkie ale nie pokolei
			//ten button wywoluje gaxes.cmd.home
			IF gAxes.Ctrl.MpTransporterAxis.IsHomed AND gAxes.Ctrl.MpCartAxis.IsHomed AND gAxes.Ctrl.MpPourerAxis.IsHomed THEN
				//ustawiamy odpowiedni layer
				Machine.States.MachineState:=STATE_WAIT_FOR_CMD_MACHINE;
			END_IF;
		//zamiast main moze wait for cmd?
		STATE_WAIT_FOR_CMD_MACHINE:
			IF EDGEPOS(Machine.Cmd.MachineCmd.Start) THEN
				Machine.Cmd.MachineCmd.Start:=FALSE;
				Machine.States.MachineState:=STATE_START_MACHINE;
				//odpowiedni layer, powinien bych chyba ten co w init
			END_IF;
			IF EDGEPOS(Machine.Cmd.MachineCmd.Stop) THEN
				//stop layer -> pokazuja sie przyciski od home kazdej osi
				Machine.Cmd.MachineCmd.Stop:=FALSE;
				Machine.States.MachineState:=STATE_STOP_MACHINE;
			END_IF;
			IF EDGEPOS(Machine.Cmd.MachineCmd.ManualCtrl) THEN
				Machine.Cmd.MachineCmd.ManualCtrl:=FALSE;
				Machine.States.MachineState:=STATE_MANUAL_MACHINE;
			END_IF
			IF EDGEPOS(Machine.Cmd.MachineCmd.AutoCtrl) THEN
				Machine.Cmd.MachineCmd.AutoCtrl:=FALSE;
				Machine.States.MachineState:=STATE_AUTO_MACHINE;
			END_IF
			MachineAxesPosition.Tasma:=gAxes.Ctrl.MpTransporterAxis.Position;
			MachineAxesPosition.Wozek:=gAxes.Ctrl.MpCartAxis.Position;
			MachineAxesPosition.Nalewak:=gAxes.Ctrl.MpPourerAxis.Position;
			AdrAxesPositions:=ADR(MachineAxesPosition);
			Machine.GUI.uiShowLayer[0]:=1; //strona glowna
		STATE_START_MACHINE:
			//layer taki jak w home
			gAxes.Cmd.Auto.MoveVelocity:=TRUE;
			Machine.States.MachineState:=STATE_WAIT_FOR_CMD_MACHINE;
			//wylaczenie odpowiednich leyerow
		STATE_STOP_MACHINE:
			gAxes.Ctrl.MpTransporterAxis.MoveVelocity:=FALSE;
			Machine.States.MachineState:=STATE_WAIT_FOR_CMD_MACHINE;
			//wlaczenie layeru w ktorym sa podlaczone przyciski z komendami hommowania
		STATE_MANUAL_MACHINE:
			IF gAxes.Ctrl.MpTransporterAxis.MoveActive THEN
				Machine.States.MachineState:=STATE_WAIT_FOR_CMD_MACHINE;
				//alarm maszyna w ruchu nie mozesz przejsc do tryby manualnego
			ELSE
				gAxes.SequencerCtrl.MpAxisCamSequencer_0.StartSequence:=FALSE;
				gAxes.SequencerCtrl.MpAxisCamSequencer_1.StartSequence:=FALSE;
				//pojawiaja sie przyciski od jog
				Machine.States.MachineState:=STATE_WAIT_FOR_CMD_MACHINE;
			END_IF;
		STATE_AUTO_MACHINE:
//			IF gAxes.Ctrl.MpTransporterAxis.MoveActive OR gAxes.Ctrl.MpTransporterAxis.MoveActive THEN
//	  			zabezpieczenie ze jesli jetw ruchu to nie mozna z manual do auto
			//			END_IF;
			IF gAxes.Ctrl.MpPourerAxis.Position <> 0 THEN
				gAxes.Ctrl.MpPourerAxis.MoveAbsolute:=TRUE;
			ELSE
				gAxes.Ctrl.MpPourerAxis.MoveAbsolute:=FALSE;
			END_IF

			IF gAxes.Ctrl.MpCartAxis.Position <> 0 AND gAxes.Ctrl.MpPourerAxis.Position=0 THEN
				gAxes.Ctrl.MpCartAxis.MoveAbsolute:=TRUE;
			ELSE
				gAxes.Ctrl.MpCartAxis.MoveAbsolute:=FALSE;
			END_IF

			IF gAxes.Ctrl.MpPourerAxis.Position=0 AND gAxes.Ctrl.MpCartAxis.Position=0 THEN
				gAxes.Ctrl.MpTransporterAxisPar.Position:=gAxes.Ctrl.MpTransporterAxis.Position+(500-brmfmod(LREAL_TO_REAL(gAxes.Ctrl.MpTransporterAxis.Position),500))+500;
				gAxes.Cmd.Auto.Update:=TRUE;
				gAxes.Ctrl.MpTransporterAxis.MoveAbsolute:=TRUE;
			END_IF

		//next case to wait for cmd

	END_CASE;

//	Machine.SequencerCtrl.MpAxisCamSequencer_0.MpLink:=ADR(gCartAxisCfg);
//	Machine.SequencerCtrl.MpAxisCamSequencer_0.MpLinkMaster:=ADR(gTranAxisCfg);
//	Machine.SequencerCtrl.MpAxisCamSequencer_0.Parameters:=ADR(Machine.SequencerCtrl.MpAxisCamSequencerPar_0);
//	Machine.SequencerCtrl.MpAxisCamSequencer_0();

	//	Machine.SequencerCtrl.MpAxisCamSequencer_1.MpLink:=ADR(gPourAxisCfg);
	//	Machine.SequencerCtrl.MpAxisCamSequencer_1.MpLinkMaster:=ADR(gCartAxisCfg);
	//	Machine.SequencerCtrl.MpAxisCamSequencer_1.Parameters:=ADR(Machine.SequencerCtrl.MpAxisCamSequencerPar_1);
//	//Machine.SequencerCtrl.MpAxisCamSequencer_1.Signal1:=Machine.SequencerCtrl.MpAxisCamSequencer_0.InCompensation;
//	Machine.SequencerCtrl.MpAxisCamSequencer_1();
END_PROGRAM

PROGRAM _EXIT
	(* Insert code here *)

END_PROGRAM
```

### GlobalMachine.typ
```iecst
(* AutoAxis *)
TYPE
	gAxesCtrlType : 	STRUCT
		Ctrl : gAxisBasicCtrlType;
		SequencerCtrl : gAxisCamSequencerType;
		Cmd : gCmdType;
		State : gStateType;
		Timers : gTimersType;
		TimersPar : gTimersParType;
	END_STRUCT;
	gAxisCamSequencerType : STRUCT
		MpAxisCamSequencer_0 : MpAxisCamSequencer;
		MpAxisCamSequencerPar_0 : MpAxisCamSequencerParType;
		MpAxisCamSequencer_1 : MpAxisCamSequencer;
		MpAxisCamSequencerPar_1 : MpAxisCamSequencerParType;
	END_STRUCT;
	gAxisBasicCtrlType : 	STRUCT
		MpTransporterAxis : MpAxisBasic;
		MpTransporterAxisPar : MpAxisBasicParType;
		MpCartAxis : MpAxisBasic;
		MpCartAxisPar : MpAxisBasicParType;
		MpPourerAxis : MpAxisBasic;
		MpPourerAxisPar : MpAxisBasicParType;
	END_STRUCT;
	gCmdType : 	STRUCT
		Auto : gAutoCmdType;
		Manual : gManualCmdType;
	END_STRUCT;

	gAutoCmdType : STRUCT
		Power : BOOL;
		Home : BOOL;
		Update : BOOL;
		Stop : BOOL;
		ErrorReset : BOOL;
		MoveVelocity : BOOL;
		MoveAdditive : BOOL;
		MoveAbsolute : BOOL;
	END_STRUCT;

	gManualCmdType : STRUCT
		TransporterJogPositive : BOOL;
		TransporterJogNegative : BOOL;
		CartJogPositive : BOOL;
		CartJogNegative : BOOL;
		PourerJogPositive : BOOL;
		PourerJogNegative : BOOL;

		TransporterHomming : BOOL;
		CartHomming : BOOL;
		PourerHomming : BOOL;
	END_STRUCT;

	gTimersType : STRUCT
		PowerTimer : ARRAY[0..2] OF TON;
		HomeTimer : ARRAY[0..2] OF TON;
	END_STRUCT;

	gTimersParType : STRUCT
		PowerDelayTime : REAL :=5;
		HomeDelayTime : REAL :=5;
	END_STRUCT;

	gStateType : STRUCT
		Auto : gAutoAxisStateType;
		Manual : gManualAxisStateType;
	END_STRUCT;

	gAutoAxisStateType :
		(
		STATE_INIT_AXES := 0,
		STATE_WAIT_FOR_CMD_AXES := 1,
		STATE_POWER_ON_AXES := 2,
		STATE_HOME_AXES := 3,
		STATE_UPDATE_AXES := 4,
		STATE_MOVE_VELOCITY_AXES := 5,
		STATE_MOVE_ABSOLUTE_AXES := 6,
		STATE_MOVE_ADDITIVE_AXES := 7,
		STATE_STOP_AXES := 8,
		STATE_ERROR_AXES := 10
	);

	gManualAxisStateType :
		(
		STATE_WAIT_FOR_CMD_MANUAL := 0,
		STATE_TRANSPORTER_HOMMING :=1,
		STATE_CART_HOMMING :=2,
		STATE_POURER_HOMMING :=3
	);
END_TYPE
```

### GlobalMachine.var
```iecst
VAR
	gControlType : BOOL;
	gAxes : gAxesCtrlType;
END_VAR

VAR CONSTANT

END_VAR
```

### Program Logical/Software/Code/AlarmControl/AlarmCtrl

#### Types.typ
```iecst
TYPE
	AlarmCtrlType : STRUCT
		AlarmBasic : MpAlarmBasic;
		AlarmBasicUI : MpAlarmBasicUI;
		UserAlarmBasicUI : MpAlarmBasicUI;
		RecipeAlarmBasicUI : MpAlarmBasicUI;
		MyAlarmBasicUI : MpAlarmBasicUI;

		AlarmRegUser : MpAlarmRegUser;

		RecipeAlarm : MpAlarmBasicUIConnect20Type;
		AxisAlarm : MpAlarmBasicUIConnect20Type;
		UserAlarm : MpAlarmBasicUIConnect20Type;
		MyAlarm : MpAlarmBasicUIConnect20Type;
	END_STRUCT;
END_TYPE
```

#### Variables.var
```iecst
VAR
	Alarm : AlarmCtrlType;
END_VAR

VAR CONSTANT

END_VAR
```

#### Main.st
```iecst
PROGRAM _INIT
	(* Insert code here *)
	Alarm.AlarmBasic.Enable:=TRUE;
	Alarm.AlarmBasicUI.Enable:=TRUE;
	Alarm.UserAlarmBasicUI.Enable:=TRUE;
	Alarm.RecipeAlarmBasicUI.Enable:=TRUE;
	Alarm.MyAlarmBasicUI.Enable:=TRUE;
	Alarm.AlarmRegUser.Enable:=TRUE;
END_PROGRAM

PROGRAM _CYCLIC
	(* Insert code here *)
	Alarm.AlarmBasic.MpLink:=ADR(gAlarmBasic);
	Alarm.AlarmBasicUI.MpLink:=ADR(gTranAxisCfg);
	Alarm.UserAlarmBasicUI.MpLink:=ADR(gUserLogin);
	Alarm.RecipeAlarmBasicUI.MpLink:=ADR(gRecipeXml);

	Alarm.AlarmBasicUI.Mode:=mpALARM_BASIC_UI_MODE_ALL;
	Alarm.AlarmBasicUI.UISetup.AcknowledgeImage:=ADR(Alarm.AxisAlarm.AcknowledgeImage[0]);
	Alarm.AlarmBasicUI.UISetup.AlarmImage:=ADR(Alarm.AxisAlarm.AlarmImage[0]);
	Alarm.AlarmBasicUI.UISetup.ImageSize:=SIZEOF(Alarm.AxisAlarm.AlarmImage)/SIZEOF(Alarm.AxisAlarm.AlarmImage[0]);
	Alarm.AlarmBasicUI.UISetup.AddInfo:=ADR(Alarm.AxisAlarm.AddInfo[0]);
	Alarm.AlarmBasicUI.UISetup.AddInfoStringSize:=SIZEOF(Alarm.AxisAlarm.AddInfo[0]);

	Alarm.UserAlarmBasicUI.Mode:=mpALARM_BASIC_UI_MODE_ALL;
	Alarm.UserAlarmBasicUI.UISetup.AcknowledgeImage:=ADR(Alarm.UserAlarm.AcknowledgeImage[0]);
	Alarm.UserAlarmBasicUI.UISetup.AlarmImage:=ADR(Alarm.UserAlarm.AlarmImage[0]);
	Alarm.UserAlarmBasicUI.UISetup.ImageSize:=SIZEOF(Alarm.UserAlarm.AlarmImage)/SIZEOF(Alarm.UserAlarm.AlarmImage[0]);
	Alarm.UserAlarmBasicUI.UISetup.AddInfo:=ADR(Alarm.UserAlarm.AddInfo[0]);
	Alarm.UserAlarmBasicUI.UISetup.AddInfoStringSize:=SIZEOF(Alarm.UserAlarm.AddInfo[0]);

	Alarm.RecipeAlarmBasicUI.Mode:=mpALARM_BASIC_UI_MODE_ALL;
	Alarm.RecipeAlarmBasicUI.UISetup.AcknowledgeImage:=ADR(Alarm.RecipeAlarm.AcknowledgeImage[0]);
	Alarm.RecipeAlarmBasicUI.UISetup.AlarmImage:=ADR(Alarm.RecipeAlarm.AlarmImage[0]);
	Alarm.RecipeAlarmBasicUI.UISetup.ImageSize:=SIZEOF(Alarm.RecipeAlarm.AlarmImage)/SIZEOF(Alarm.RecipeAlarm.AlarmImage[0]);
	Alarm.RecipeAlarmBasicUI.UISetup.AddInfo:=ADR(Alarm.RecipeAlarm.AddInfo[0]);
	Alarm.RecipeAlarmBasicUI.UISetup.AddInfoStringSize:=SIZEOF(Alarm.RecipeAlarm.AddInfo[0]);

	Alarm.MyAlarmBasicUI.MpLink:=ADR(gAlarmBasic);
	Alarm.MyAlarmBasicUI.Mode:=mpALARM_BASIC_UI_MODE_USER;
	Alarm.MyAlarmBasicUI.UISetup.AcknowledgeImage:=ADR(Alarm.MyAlarm.AcknowledgeImage[0]);
	Alarm.MyAlarmBasicUI.UISetup.AlarmImage:=ADR(Alarm.MyAlarm.AlarmImage[0]);
	Alarm.MyAlarmBasicUI.UISetup.ImageSize:=SIZEOF(Alarm.MyAlarm.AlarmImage)/SIZEOF(Alarm.MyAlarm.AlarmImage[0]);
	Alarm.MyAlarmBasicUI.UISetup.AddInfo:=ADR(Alarm.MyAlarm.AddInfo[0]);
	Alarm.MyAlarmBasicUI.UISetup.AddInfoStringSize:=SIZEOF(Alarm.MyAlarm.AddInfo[0]);

	Alarm.AlarmRegUser.MpLink:=ADR(gAlarmBasic);
	Alarm.AlarmRegUser.NumberOfAlarms:=2;
	//Alarm.AlarmRegUser.mode

	//Alarm.

	Alarm.AlarmBasic();
	Alarm.AlarmBasicUI();
	Alarm.UserAlarmBasicUI();
	Alarm.RecipeAlarmBasicUI();
	Alarm.AlarmRegUser();
	Alarm.MyAlarmBasicUI();
END_PROGRAM

PROGRAM _EXIT
	(* Insert code here *)

END_PROGRAM
```

### Program Logical/Software/Code/AutoAxisCtrl

#### Main.st
```iecst
PROGRAM _INIT
	(* Insert code here *)
	(* To DO -> timer w homming, brak wylaczania zasilani *)
	gAxes.State:=STATE_INIT_AXES;
	gControlType:=TRUE;
END_PROGRAM

PROGRAM _CYCLIC
	(* Insert code here *)
	gAxes.Ctrl.MpTransporterAxis.MpLink:=ADR(gTranAxisCfg);
	gAxes.Ctrl.MpTransporterAxis.Parameters:=ADR(gAxes.Ctrl.MpTransporterAxisPar);
	gAxes.Ctrl.MpTransporterAxis.Axis:=ADR(gTranAxis);

	gAxes.Ctrl.MpCartAxis.MpLink:=ADR(gCartAxisCfg);
	gAxes.Ctrl.MpCartAxis.Parameters:=ADR(gAxes.Ctrl.MpCartAxisPar);
	gAxes.Ctrl.MpCartAxis.Axis:=ADR(gCartAxis);

	gAxes.Ctrl.MpPourerAxis.MpLink:=ADR(gPourAxisCfg);
	gAxes.Ctrl.MpPourerAxis.Parameters:=ADR(gAxes.Ctrl.MpPourerAxisPar);
	gAxes.Ctrl.MpPourerAxis.Axis:=ADR(gPourAxis);

	gAxes.Ctrl.MpTransporterAxis();
	gAxes.Ctrl.MpCartAxis();
	gAxes.Ctrl.MpPourerAxis();

	//gStateAutoAxisCtrl:=ADR(gAxes.State);
	//gCmdAutoAxisCtrl:=ADR(gAxes.Cmd);
	//CmdFromMachine ACCESS gCmdAutoAxisCtrl;
	//gAxes.Cmd:=CmdFromMachine;

	IF gControlType THEN
		IF gAxes.Ctrl.MpTransporterAxis.Error THEN
			//alarm osi transporter
			gAxes.State:=STATE_ERROR_AXES;
		END_IF
		IF gAxes.Ctrl.MpCartAxis.Error THEN
			//alarm osi wozka
			gAxes.State:=STATE_ERROR_AXES;
		END_IF
		IF gAxes.Ctrl.MpPourerAxis.Error THEN
			//alarm nalewaka
			gAxes.State:=STATE_ERROR_AXES;
		END_IF

		CASE gAxes.State OF
			STATE_INIT_AXES:
				gAxes.Ctrl.MpTransporterAxis.Enable:=TRUE;
				gAxes.Ctrl.MpCartAxis.Enable:=TRUE;
				gAxes.Ctrl.MpPourerAxis.Enable:=TRUE;

				IF gAxes.Ctrl.MpTransporterAxis.Active AND gAxes.Ctrl.MpCartAxis.Active AND gAxes.Ctrl.MpPourerAxis.Active THEN
					gAxes.State:=STATE_POWER_ON_AXES;
				END_IF;
			STATE_WAIT_FOR_CMD_AXES:
				IF EDGEPOS(gAxes.Cmd.Power) THEN
					gAxes.Cmd.Power:=FALSE;
					gAxes.State:=STATE_POWER_ON_AXES;
				ELSIF EDGEPOS(gAxes.Cmd.Home) THEN
					gAxes.Cmd.Home:=FALSE;
					gAxes.State:=STATE_HOME_AXES;
				ELSIF EDGEPOS(gAxes.Cmd.Update) THEN
					gAxes.Cmd.Update:=FALSE;
					gAxes.State:=STATE_UPDATE_AXES;
				ELSIF EDGEPOS(gAxes.Cmd.Stop) THEN
					gAxes.Cmd.Stop:=FALSE;
					gAxes.State:=STATE_STOP_AXES;
				ELSIF EDGEPOS(gAxes.Cmd.ErrorReset) THEN
					gAxes.Cmd.ErrorReset:=FALSE;

				ELSIF EDGEPOS(gAxes.Cmd.MoveVelocity) THEN
					gAxes.Cmd.MoveVelocity:=FALSE;
					gAxes.State:=STATE_MOVE_VELOCITY_AXES;
//				ELSIF gAxes.Cmd.MoveAbsolute THEN
//				ELSIF gAxes.Cmd.MoveAdditive THEN
				END_IF;
			STATE_POWER_ON_AXES:
				gAxes.Ctrl.MpTransporterAxis.Power:=TRUE;
				gAxes.Ctrl.MpCartAxis.Power:=TRUE;
				gAxes.Ctrl.MpPourerAxis.Power:=TRUE;

				gAxes.Timers.PowerTimer[0].IN:=NOT(gAxes.Ctrl.MpTransporterAxis.PowerOn);
				gAxes.Timers.PowerTimer[0].PT:=REAL_TO_TIME(gAxes.TimersPar.PowerDelayTime*1000);
				gAxes.Timers.PowerTimer[0]();

				gAxes.Timers.PowerTimer[1].IN:=NOT(gAxes.Ctrl.MpCartAxis.PowerOn);
				gAxes.Timers.PowerTimer[1].PT:=REAL_TO_TIME(gAxes.TimersPar.PowerDelayTime*1000);
				gAxes.Timers.PowerTimer[1]();

				gAxes.Timers.PowerTimer[2].IN:=NOT(gAxes.Ctrl.MpPourerAxis.PowerOn);
				gAxes.Timers.PowerTimer[2].PT:=REAL_TO_TIME(gAxes.TimersPar.PowerDelayTime*1000);
				gAxes.Timers.PowerTimer[2]();

				IF gAxes.Timers.PowerTimer[0].Q THEN
					//zbyt dlugie zalaczanie osi transportra alarm
					gAxes.Timers.PowerTimer[0].IN:=FALSE;
					gAxes.Timers.PowerTimer[0]();
					gAxes.State:=STATE_ERROR_AXES;
				END_IF;
				IF gAxes.Timers.PowerTimer[1].Q THEN
					//zbyt dlugie zalaczanie osi wozka alarm
					gAxes.Timers.PowerTimer[1].IN:=FALSE;
					gAxes.Timers.PowerTimer[1]();
					gAxes.State:=STATE_ERROR_AXES;
				END_IF;
				IF gAxes.Timers.PowerTimer[2].Q THEN
					//zbyt dlugie zalaczanie osi nalewaka alarm
					gAxes.Timers.PowerTimer[2].IN:=FALSE;
					gAxes.Timers.PowerTimer[2]();
					gAxes.State:=STATE_ERROR_AXES;
				END_IF;

				IF gAxes.Ctrl.MpTransporterAxis.PowerOn AND gAxes.Ctrl.MpCartAxis.PowerOn AND gAxes.Ctrl.MpPourerAxis.PowerOn THEN
					gAxes.State:=STATE_WAIT_FOR_CMD_AXES;
					gAxes.Timers.PowerTimer[0].IN:=FALSE;
					gAxes.Timers.PowerTimer[0]();
					gAxes.Timers.PowerTimer[1].IN:=FALSE;
					gAxes.Timers.PowerTimer[1]();
					gAxes.Timers.PowerTimer[2].IN:=FALSE;
					gAxes.Timers.PowerTimer[2]();
				END_IF;

			STATE_HOME_AXES:
				gAxes.Ctrl.MpTransporterAxis.Home:=TRUE;
				gAxes.Ctrl.MpCartAxis.Home:=TRUE;
				gAxes.Ctrl.MpPourerAxis.Home:=TRUE;

				gAxes.Timers.HomeTimer[0].IN:=NOT(gAxes.Ctrl.MpTransporterAxis.IsHomed);
				gAxes.Timers.HomeTimer[0].PT:=REAL_TO_TIME(gAxes.TimersPar.HomeDelayTime*1000);
				gAxes.Timers.HomeTimer[0]();

				gAxes.Timers.HomeTimer[1].IN:=NOT(gAxes.Ctrl.MpCartAxis.IsHomed);
				gAxes.Timers.HomeTimer[1].PT:=REAL_TO_TIME(gAxes.TimersPar.HomeDelayTime*1000);
				gAxes.Timers.HomeTimer[1]();

				gAxes.Timers.HomeTimer[2].IN:=NOT(gAxes.Ctrl.MpPourerAxis.IsHomed);
				gAxes.Timers.HomeTimer[2].PT:=REAL_TO_TIME(gAxes.TimersPar.HomeDelayTime*1000);
				gAxes.Timers.HomeTimer[2]();

				IF gAxes.Timers.HomeTimer[0].Q THEN
					gAxes.Timers.HomeTimer[0].IN:=FALSE;
					gAxes.Timers.HomeTimer[0]();
					//zbyt dlugie bazowanie osi transportra alarm
					gAxes.State:=STATE_ERROR_AXES;
				END_IF;

				IF gAxes.Timers.HomeTimer[1].Q THEN
					gAxes.Timers.HomeTimer[1].IN:=FALSE;
					gAxes.Timers.HomeTimer[1]();
					//zbyt dlugie bazowanie osi wozka alarm
					gAxes.State:=STATE_ERROR_AXES;
				END_IF;

				IF gAxes.Timers.HomeTimer[2].Q THEN
					gAxes.Timers.HomeTimer[2].IN:=FALSE;
					gAxes.Timers.HomeTimer[2]();
					//zbyt dlugie bazowanie osi nalewaka alarm
					gAxes.State:=STATE_ERROR_AXES;
				END_IF;

				IF gAxes.Ctrl.MpTransporterAxis.IsHomed AND gAxes.Ctrl.MpCartAxis.IsHomed AND gAxes.Ctrl.MpPourerAxis.IsHomed THEN
					gAxes.Ctrl.MpTransporterAxis.Home:=FALSE;
					gAxes.Ctrl.MpCartAxis.Home:=FALSE;
					gAxes.Ctrl.MpPourerAxis.Home:=FALSE;
					gAxes.State:=STATE_WAIT_FOR_CMD_AXES;
					gAxes.Timers.HomeTimer[0].IN:=FALSE;
					gAxes.Timers.HomeTimer[0]();
					gAxes.Timers.HomeTimer[1].IN:=FALSE;
					gAxes.Timers.HomeTimer[1]();
					gAxes.Timers.HomeTimer[2].IN:=FALSE;
					gAxes.Timers.HomeTimer[2]();
				END_IF;
			STATE_STOP_AXES:
				//bez wylaczania zasialania
				(* Sprawdzenie czy jes wlaczonysilnik jesi tak to stop - jesli off to wywalierror *)
				IF gAxes.Ctrl.MpTransporterAxis.PowerOn THEN
					gAxes.Ctrl.MpTransporterAxis.Stop:=TRUE;
				END_IF;

				IF gAxes.Ctrl.MpCartAxis.PowerOn THEN
					gAxes.Ctrl.MpCartAxis.Stop:=TRUE;
				END_IF;

				IF gAxes.Ctrl.MpPourerAxis.PowerOn THEN
					gAxes.Ctrl.MpPourerAxis.Stop:=TRUE;
				END_IF;

				IF gAxes.Ctrl.MpTransporterAxis.Stopped AND gAxes.Ctrl.MpCartAxis.Stopped AND gAxes.Ctrl.MpPourerAxis.Stopped THEN

					gAxes.Ctrl.MpTransporterAxis.Stop:=FALSE;
					gAxes.Ctrl.MpCartAxis.Stop:=FALSE;
					gAxes.Ctrl.MpPourerAxis.Stop:=FALSE;

					gAxes.Ctrl.MpTransporterAxis.MoveVelocity:=FALSE;

					gAxes.State:=STATE_WAIT_FOR_CMD_AXES;
					//gAxes.Cmd.Stop:=FALSE;
				END_IF;
			STATE_UPDATE_AXES:
				gAxes.Ctrl.MpTransporterAxis.Update:=TRUE;
				gAxes.Ctrl.MpCartAxis.Update:=TRUE;
				gAxes.Ctrl.MpPourerAxis.Update:=TRUE;

				IF gAxes.Ctrl.MpTransporterAxis.UpdateDone AND gAxes.Ctrl.MpCartAxis.UpdateDone AND gAxes.Ctrl.MpPourerAxis.UpdateDone THEN
					gAxes.State:=STATE_WAIT_FOR_CMD_AXES;
					gAxes.Ctrl.MpTransporterAxis.Update:=FALSE;
					gAxes.Ctrl.MpCartAxis.Update:=FALSE;
					gAxes.Ctrl.MpPourerAxis.Update:=FALSE;
				END_IF;
			STATE_MOVE_VELOCITY_AXES:
				(* Chyba że tu tdac ze ready  *)
				gAxes.Ctrl.MpTransporterAxis.MoveVelocity:=TRUE;
				gAxes.State:=STATE_WAIT_FOR_CMD_AXES;
			STATE_ERROR_AXES:
				(* Zatrzymanie wszystkich silnikow *)
				gAxes.Ctrl.MpTransporterAxis.MoveVelocity:=FALSE;
				IF gAxes.Ctrl.MpTransporterAxis.PowerOn THEN
					gAxes.Ctrl.MpTransporterAxis.Stop:=TRUE;
				END_IF;

				IF gAxes.Ctrl.MpCartAxis.PowerOn THEN
					gAxes.Ctrl.MpCartAxis.Stop:=TRUE;
				END_IF;

				IF gAxes.Ctrl.MpPourerAxis.PowerOn THEN
					gAxes.Ctrl.MpPourerAxis.Stop:=TRUE;
				END_IF;

				(* Jesli sa zastopowane to power off  *)
				IF gAxes.Ctrl.MpTransporterAxis.Stopped THEN
					gAxes.Ctrl.MpTransporterAxis.Power:=FALSE;
				END_IF;

				IF gAxes.Ctrl.MpCartAxis.Stopped THEN
					gAxes.Ctrl.MpCartAxis.Power:=FALSE;
				END_IF;

				IF gAxes.Ctrl.MpPourerAxis.Stopped THEN
					gAxes.Ctrl.MpPourerAxis.Power:=FALSE;
				END_IF;

				(* Czekamy na przycisk reseterror *)
				IF EDGEPOS(gAxes.Cmd.ErrorReset) AND (NOT(gAxes.Ctrl.MpTransporterAxis.PowerOn) AND NOT(gAxes.Ctrl.MpCartAxis.PowerOn) AND NOT(gAxes.Ctrl.MpPourerAxis.PowerOn)) THEN
					gAxes.Cmd.ErrorReset:=FALSE;

					gAxes.Ctrl.MpTransporterAxis.Stop:=FALSE;
					gAxes.Ctrl.MpCartAxis.Stop:=FALSE;
					gAxes.Ctrl.MpPourerAxis.Stop:=FALSE;

					gAxes.Ctrl.MpTransporterAxis.ErrorReset:=TRUE;
					gAxes.Ctrl.MpCartAxis.ErrorReset:=TRUE;
					gAxes.Ctrl.MpPourerAxis.ErrorReset:=TRUE;
					//gAxes.State:=WAIT_FOR_CMD;
				END_IF;

				IF NOT(gAxes.Ctrl.MpTransporterAxis.Error) AND NOT(gAxes.Ctrl.MpCartAxis.Error) AND NOT(gAxes.Ctrl.MpPourerAxis.Error) THEN
					gAxes.Ctrl.MpTransporterAxis.ErrorReset:=FALSE;
					gAxes.Ctrl.MpCartAxis.ErrorReset:=FALSE;
					gAxes.Ctrl.MpPourerAxis.ErrorReset:=FALSE;
					gAxes.State:=STATE_WAIT_FOR_CMD_AXES;
					//gAxes.Ctrl.MpTransporterAxis.MoveVelocity:=FALSE;
				END_IF

		END_CASE;
	END_IF;

END_PROGRAM

PROGRAM _EXIT
	(* Insert code here *)
	gAxes.Ctrl.MpTransporterAxis.Power:=FALSE;
	gAxes.Ctrl.MpTransporterAxis.Enable:=FALSE;
	gAxes.Ctrl.MpTransporterAxis();

	gAxes.Ctrl.MpCartAxis.Power:=FALSE;
	gAxes.Ctrl.MpCartAxis.Enable:=FALSE;
	gAxes.Ctrl.MpCartAxis();

	gAxes.Ctrl.MpPourerAxis.Power:=FALSE;
	gAxes.Ctrl.MpPourerAxis.Enable:=FALSE;
	gAxes.Ctrl.MpPourerAxis();

END_PROGRAM
```

### AxisCtrlGlobal.typ
```iecst
(* AutoAxis *)

TYPE
	(* Główny typ zawierający inne typy *)
	gAxesCtrlType : 	STRUCT
		Ctrl : gAxisBasicCtrlType;
		Cmd : gCmdType;
		State : gStateType;
		Timers : gTimersType;
		TimersPar : gTimersParType;
	END_STRUCT;
	(* Typ zawierający bloki mpAxisBasic *)
	gAxisBasicCtrlType : 	STRUCT
		MpTransporterAxis : MpAxisBasic;
		MpTransporterAxisPar : MpAxisBasicParType;
		MpCartAxis : MpAxisBasic;
		MpCartAxisPar : MpAxisBasicParType;
		MpPourerAxis : MpAxisBasic;
		MpPourerAxisPar : MpAxisBasicParType;
	END_STRUCT;
	(* Główny typ komend  *)
	gCmdType : 	STRUCT
		Auto : gAutoCmdType;
		Manual : gManualCmdType;
	END_STRUCT;
	(* Typ zawierający komendy sterujący silnikami w trybie automatycznym *)
	gAutoCmdType : 	STRUCT
		Power : BOOL;
		Home : BOOL;
		Update : BOOL;
		Stop : BOOL;
		ErrorReset : BOOL;
		MoveVelocity : BOOL;
	END_STRUCT;
	(* Typ zawierający komdendy do sterowania manualnego *)
	gManualCmdType : 	STRUCT
		TransporterHomming : BOOL;
		CartHomming : BOOL;
		PourerHomming : BOOL;
	END_STRUCT;
	gTimersType : 	STRUCT
		HomeTimer : ARRAY[0..2]OF TON;
	END_STRUCT;
	gTimersParType : 	STRUCT
		HomeDelayTime : REAL := 5;
	END_STRUCT;
	(* Główny typ zawierający stany do maszyn *)
	gStateType : 	STRUCT
		Auto : gAutoAxisStateType;
		Manual : gManualAxisStateType;
	END_STRUCT;
	gAutoAxisStateType :
		(
		STATE_INIT_AXES := 0,
		STATE_WAIT_FOR_CMD_AXES := 1,
		STATE_POWER_ON_AXES := 2,
		STATE_HOME_AXES := 3,
		STATE_UPDATE_AXES := 4,
		STATE_MOVE_VELOCITY_AXES := 5,
		STATE_STOP_AXES := 8,
		STATE_ERROR_AXES := 10
		);
	gManualAxisStateType :
		(
		STATE_WAIT_FOR_CMD_MANUAL := 0,
		STATE_TRANSPORTER_HOMMING := 1,
		STATE_CART_HOMMING := 2,
		STATE_POURER_HOMMING := 3
		);
END_TYPE
```

### AxisCtrlGlobal.var
```iecst
VAR
	gAxes : gAxesCtrlType;
	(* zmienna wykorzystywana do przekazywania pozycji do scene viewera *)
	MachineAxesPosition : AxesPositionsType;
END_VAR
```

### Program Logical/Software/Code/AxisControl/AxisCtrl

#### Main.st
```iecst
PROGRAM _INIT
	(* Insert code here *)
	gAxes.State.Auto:=STATE_INIT_AXES;
END_PROGRAM

PROGRAM _CYCLIC
	(* Insert code here *)
	gAxes.Ctrl.MpTransporterAxis.MpLink:=ADR(gTranAxisCfg);
	gAxes.Ctrl.MpTransporterAxis.Parameters:=ADR(gAxes.Ctrl.MpTransporterAxisPar);
	gAxes.Ctrl.MpTransporterAxis.Axis:=ADR(gTranAxis);

	gAxes.Ctrl.MpCartAxis.MpLink:=ADR(gCartAxisCfg);
	gAxes.Ctrl.MpCartAxis.Parameters:=ADR(gAxes.Ctrl.MpCartAxisPar);
	gAxes.Ctrl.MpCartAxis.Axis:=ADR(gCartAxis);

	gAxes.Ctrl.MpPourerAxis.MpLink:=ADR(gPourAxisCfg);
	gAxes.Ctrl.MpPourerAxis.Parameters:=ADR(gAxes.Ctrl.MpPourerAxisPar);
	gAxes.Ctrl.MpPourerAxis.Axis:=ADR(gPourAxis);

	(* Warunki sprawdzające na której osi występuje error *)
	IF gAxes.Ctrl.MpTransporterAxis.Error THEN
		//alarm osi transporter
		gAxes.State.Auto:=STATE_ERROR_AXES;
	END_IF
	IF gAxes.Ctrl.MpCartAxis.Error THEN
		//alarm osi wozka
		gAxes.State.Auto:=STATE_ERROR_AXES;
	END_IF
	IF gAxes.Ctrl.MpPourerAxis.Error THEN
		//alarm nalewaka
		gAxes.State.Auto:=STATE_ERROR_AXES;
	END_IF

	(* Główna maszyna stanów osi *)
	CASE gAxes.State.Auto OF
		(* Stan inicjalizacyjny -> uruchomienie bloków, podstawowe parametry, przejscie dalej *)
		STATE_INIT_AXES:
			//MpAlarmSet(gAlarmBasic,0,'k');
			gAxes.Ctrl.MpTransporterAxis.Enable:=TRUE;
			gAxes.Ctrl.MpCartAxis.Enable:=TRUE;
			gAxes.Ctrl.MpPourerAxis.Enable:=TRUE;

			gAxes.Ctrl.MpTransporterAxisPar.Acceleration:=500;
			gAxes.Ctrl.MpCartAxisPar.Acceleration:=500;
			gAxes.Ctrl.MpPourerAxisPar.Acceleration:=500;

			gAxes.Ctrl.MpTransporterAxisPar.Deceleration:=500;
			gAxes.Ctrl.MpCartAxisPar.Deceleration:=500;
			gAxes.Ctrl.MpPourerAxisPar.Deceleration:=500;

			gAxes.Ctrl.MpTransporterAxisPar.Velocity:=100;
			gAxes.Ctrl.MpCartAxisPar.Velocity:=100;
			gAxes.Ctrl.MpPourerAxisPar.Velocity:=100;

			(* Jesli bloki aktywne przejdz do włączenia zasilania *)
			IF gAxes.Ctrl.MpTransporterAxis.Active AND gAxes.Ctrl.MpCartAxis.Active AND gAxes.Ctrl.MpPourerAxis.Active THEN
				gAxes.State.Auto:=STATE_POWER_ON_AXES;
			END_IF;
		STATE_WAIT_FOR_CMD_AXES:
			IF EDGEPOS(gAxes.Cmd.Auto.Power) THEN
				gAxes.Cmd.Auto.Power:=FALSE;
				gAxes.State.Auto:=STATE_POWER_ON_AXES;
			ELSIF EDGEPOS(gAxes.Cmd.Auto.Home) THEN
				gAxes.Cmd.Auto.Home:=FALSE;
				gAxes.State.Auto:=STATE_HOME_AXES;
			ELSIF EDGEPOS(gAxes.Cmd.Auto.Update) THEN
				gAxes.Cmd.Auto.Update:=FALSE;
				gAxes.State.Auto:=STATE_UPDATE_AXES;
			ELSIF EDGEPOS(gAxes.Cmd.Auto.Stop) THEN
				gAxes.Cmd.Auto.Stop:=FALSE;
				gAxes.State.Auto:=STATE_STOP_AXES;
			ELSIF EDGEPOS(gAxes.Cmd.Auto.ErrorReset) THEN
				gAxes.Cmd.Auto.ErrorReset:=FALSE;
			ELSIF EDGEPOS(gAxes.Cmd.Auto.MoveVelocity) THEN
				gAxes.Cmd.Auto.MoveVelocity:=FALSE;
				gAxes.State.Auto:=STATE_MOVE_VELOCITY_AXES;
			END_IF;
		STATE_POWER_ON_AXES:
			gAxes.Ctrl.MpTransporterAxis.Power:=TRUE;
			gAxes.Ctrl.MpCartAxis.Power:=TRUE;
			gAxes.Ctrl.MpPourerAxis.Power:=TRUE;

			IF gAxes.Ctrl.MpTransporterAxis.PowerOn AND gAxes.Ctrl.MpCartAxis.PowerOn AND gAxes.Ctrl.MpPourerAxis.PowerOn THEN
				gAxes.State.Auto:=STATE_WAIT_FOR_CMD_AXES;
			END_IF;

		STATE_HOME_AXES:
			(* Automatyczne bazowanie wszystkich osi po kolei  *)
			gAxes.Ctrl.MpTransporterAxis.Home:=TRUE;
			gAxes.Ctrl.MpCartAxis.Home:=gAxes.Ctrl.MpTransporterAxis.IsHomed;
			gAxes.Ctrl.MpPourerAxis.Home:=gAxes.Ctrl.MpCartAxis.IsHomed;

			(* Wykorzystanie zegarkow do sprawdzenia czy zadana oś została zbazowana w odpowiednim czasie *)
			gAxes.Timers.HomeTimer[0].IN:=NOT(gAxes.Ctrl.MpTransporterAxis.IsHomed);
			gAxes.Timers.HomeTimer[0].PT:=REAL_TO_TIME(gAxes.TimersPar.HomeDelayTime*1000);
			gAxes.Timers.HomeTimer[0]();

			gAxes.Timers.HomeTimer[1].IN:=gAxes.Ctrl.MpTransporterAxis.IsHomed AND NOT(gAxes.Ctrl.MpCartAxis.IsHomed);
			gAxes.Timers.HomeTimer[1].PT:=REAL_TO_TIME(gAxes.TimersPar.HomeDelayTime*1000);
			gAxes.Timers.HomeTimer[1]();

			gAxes.Timers.HomeTimer[2].IN:=gAxes.Ctrl.MpCartAxis.IsHomed AND NOT(gAxes.Ctrl.MpPourerAxis.IsHomed);
			gAxes.Timers.HomeTimer[2].PT:=REAL_TO_TIME(gAxes.TimersPar.HomeDelayTime*1000);
			gAxes.Timers.HomeTimer[2]();

			IF gAxes.Timers.HomeTimer[0].Q THEN
				gAxes.Timers.HomeTimer[0].IN:=FALSE;
				gAxes.Timers.HomeTimer[0]();
				//zbyt dlugie bazowanie osi transportra alarm
				gAxes.State.Auto:=STATE_ERROR_AXES;
			END_IF;

			IF gAxes.Timers.HomeTimer[1].Q THEN
				gAxes.Timers.HomeTimer[1].IN:=FALSE;
				gAxes.Timers.HomeTimer[1]();
				//zbyt dlugie bazowanie osi wozka alarm
				gAxes.State.Auto:=STATE_ERROR_AXES;
			END_IF;

			IF gAxes.Timers.HomeTimer[2].Q THEN
				gAxes.Timers.HomeTimer[2].IN:=FALSE;
				gAxes.Timers.HomeTimer[2]();
				//zbyt dlugie bazowanie osi nalewaka alarm
				gAxes.State.Auto:=STATE_ERROR_AXES;
			END_IF;

			(* Sprawdzenie czy wszystkie osie zostały zbazowane *)
			IF gAxes.Ctrl.MpTransporterAxis.IsHomed AND gAxes.Ctrl.MpCartAxis.IsHomed AND gAxes.Ctrl.MpPourerAxis.IsHomed THEN
				gAxes.Ctrl.MpTransporterAxis.Home:=FALSE;
				gAxes.Ctrl.MpCartAxis.Home:=FALSE;
				gAxes.Ctrl.MpPourerAxis.Home:=FALSE;
				gAxes.State.Auto:=STATE_WAIT_FOR_CMD_AXES;  //przejscie do stanu gotowosci i oczekiwanie na komendy
				gAxes.Timers.HomeTimer[0].IN:=FALSE;
				gAxes.Timers.HomeTimer[0]();
				gAxes.Timers.HomeTimer[1].IN:=FALSE;
				gAxes.Timers.HomeTimer[1]();
				gAxes.Timers.HomeTimer[2].IN:=FALSE;
				gAxes.Timers.HomeTimer[2]();
			END_IF;
		STATE_STOP_AXES:
			(* Sprawdzenie czy jes wlaczony silnik jesi tak to stop -> wywołanie .stop na wyłączonym zasilaniu generuje błąd *)
			//warning stop
			IF gAxes.Ctrl.MpTransporterAxis.PowerOn THEN
				gAxes.Ctrl.MpTransporterAxis.Stop:=TRUE;
			END_IF;

			IF gAxes.Ctrl.MpCartAxis.PowerOn THEN
				gAxes.Ctrl.MpCartAxis.Stop:=TRUE;
			END_IF;

			IF gAxes.Ctrl.MpPourerAxis.PowerOn THEN
				gAxes.Ctrl.MpPourerAxis.Stop:=TRUE;
			END_IF;

			IF gAxes.Ctrl.MpTransporterAxis.Stopped AND gAxes.Ctrl.MpCartAxis.Stopped AND gAxes.Ctrl.MpPourerAxis.Stopped THEN
				gAxes.Ctrl.MpTransporterAxis.MoveVelocity:=FALSE;
				gAxes.Ctrl.MpCartAxis.MoveVelocity:=FALSE;
				gAxes.Ctrl.MpPourerAxis.MoveVelocity:=FALSE;
				gAxes.Ctrl.MpTransporterAxis.Stop:=FALSE;
				gAxes.Ctrl.MpCartAxis.Stop:=FALSE;
				gAxes.Ctrl.MpPourerAxis.Stop:=FALSE;
				gAxes.State.Auto:=STATE_WAIT_FOR_CMD_AXES;
			END_IF;
		STATE_UPDATE_AXES:
			gAxes.Ctrl.MpTransporterAxis.Update:=TRUE;
			gAxes.Ctrl.MpCartAxis.Update:=TRUE;
			gAxes.Ctrl.MpPourerAxis.Update:=TRUE;

			IF gAxes.Ctrl.MpTransporterAxis.UpdateDone AND gAxes.Ctrl.MpCartAxis.UpdateDone AND gAxes.Ctrl.MpPourerAxis.UpdateDone THEN
				gAxes.State.Auto:=STATE_WAIT_FOR_CMD_AXES;
				gAxes.Ctrl.MpTransporterAxis.Update:=FALSE;
				gAxes.Ctrl.MpCartAxis.Update:=FALSE;
				gAxes.Ctrl.MpPourerAxis.Update:=FALSE;
			END_IF;
		STATE_MOVE_VELOCITY_AXES:
			gAxes.Ctrl.MpTransporterAxis.MoveVelocity:=TRUE;
			gAxes.State.Auto:=STATE_WAIT_FOR_CMD_AXES;
		STATE_ERROR_AXES:
			(* Zatrzymanie wszystkich silnikow *)
			gAxes.Ctrl.MpTransporterAxis.MoveVelocity:=FALSE;
			gAxes.Ctrl.MpCartAxis.MoveVelocity:=FALSE;
			gAxes.Ctrl.MpPourerAxis.MoveVelocity:=FALSE;
			gAxes.Ctrl.MpTransporterAxis.Power:=FALSE;
			gAxes.Ctrl.MpCartAxis.Power:=FALSE;
			gAxes.Ctrl.MpPourerAxis.Power:=FALSE;

			(* Czekamy na cmd reseterror *)
			IF EDGEPOS(gAxes.Cmd.Auto.ErrorReset) THEN
				gAxes.Cmd.Auto.ErrorReset:=FALSE;
				gAxes.Ctrl.MpTransporterAxis.ErrorReset:=TRUE;
				gAxes.Ctrl.MpCartAxis.ErrorReset:=TRUE;
				gAxes.Ctrl.MpPourerAxis.ErrorReset:=TRUE;
				//power na false a pozniej true do sprawdzenia
			END_IF;

			(* Jeśli wszystkie błędy zostały usunięte możemy przejść do stanu w kótrym czekamy na cmd *)
			IF NOT(gAxes.Ctrl.MpTransporterAxis.Error) AND NOT(gAxes.Ctrl.MpCartAxis.Error) AND NOT(gAxes.Ctrl.MpPourerAxis.Error) THEN
				gAxes.Ctrl.MpTransporterAxis.ErrorReset:=FALSE;
				gAxes.Ctrl.MpCartAxis.ErrorReset:=FALSE;
				gAxes.Ctrl.MpPourerAxis.ErrorReset:=FALSE;

				gAxes.Cmd.Auto.Power:=TRUE;
				gAxes.State.Auto:=STATE_WAIT_FOR_CMD_AXES;
			END_IF
	END_CASE;

	(* Maszyna stanów, ułatwiająca zarządzanie osiami w trybie manualnym *)
	CASE gAxes.State.Manual OF
		STATE_WAIT_FOR_CMD_MANUAL:
			IF EDGEPOS(gAxes.Cmd.Manual.TransporterHomming) THEN
				gAxes.Cmd.Manual.TransporterHomming:=FALSE;
				gAxes.State.Manual:=STATE_TRANSPORTER_HOMMING;
			ELSIF EDGEPOS(gAxes.Cmd.Manual.CartHomming)  THEN
				gAxes.Cmd.Manual.CartHomming:=FALSE;
				gAxes.State.Manual:=STATE_CART_HOMMING;
			ELSIF EDGEPOS(gAxes.Cmd.Manual.PourerHomming) THEN
				gAxes.Cmd.Manual.PourerHomming:=FALSE;
				gAxes.State.Manual:=STATE_POURER_HOMMING;
			END_IF;
		STATE_TRANSPORTER_HOMMING:
			gAxes.Ctrl.MpTransporterAxis.Home:=TRUE;
			gAxes.Timers.HomeTimer[0].IN:=NOT(gAxes.Ctrl.MpTransporterAxis.IsHomed);
			gAxes.Timers.HomeTimer[0].PT:=REAL_TO_TIME(gAxes.TimersPar.HomeDelayTime*1000);
			gAxes.Timers.HomeTimer[0]();

			IF gAxes.Timers.HomeTimer[0].Q THEN
				gAxes.Timers.HomeTimer[0].IN:=FALSE;
				gAxes.Timers.HomeTimer[0]();
				//zbyt dlugie bazowanie osi transportra alarm
				gAxes.State.Auto:=STATE_ERROR_AXES;
			END_IF;

			IF gAxes.Ctrl.MpTransporterAxis.IsHomed THEN
				gAxes.Ctrl.MpTransporterAxis.Home:=FALSE;
				gAxes.State.Manual:=STATE_WAIT_FOR_CMD_MANUAL;
				gAxes.Timers.HomeTimer[0].IN:=FALSE;
				gAxes.Timers.HomeTimer[0]();
			END_IF;
		STATE_CART_HOMMING:
			gAxes.Ctrl.MpCartAxis.Home:=TRUE;
			gAxes.Timers.HomeTimer[0].IN:=NOT(gAxes.Ctrl.MpCartAxis.IsHomed);
			gAxes.Timers.HomeTimer[0].PT:=REAL_TO_TIME(gAxes.TimersPar.HomeDelayTime*1000);
			gAxes.Timers.HomeTimer[0]();

			IF gAxes.Timers.HomeTimer[0].Q THEN
				gAxes.Timers.HomeTimer[0].IN:=FALSE;
				gAxes.Timers.HomeTimer[0]();
				//zbyt dlugie bazowanie osi MpCartAxis alarm
				gAxes.State.Auto:=STATE_ERROR_AXES;
			END_IF;

			IF EDGEPOS(gAxes.Ctrl.MpCartAxis.IsHomed) THEN
				gAxes.Ctrl.MpCartAxis.Home:=FALSE;
				gAxes.State.Manual:=STATE_WAIT_FOR_CMD_MANUAL;
				gAxes.Timers.HomeTimer[0].IN:=FALSE;
				gAxes.Timers.HomeTimer[0]();
			END_IF;
		STATE_POURER_HOMMING:
			gAxes.Ctrl.MpPourerAxis.Home:=TRUE;
			gAxes.Timers.HomeTimer[0].IN:=NOT(gAxes.Ctrl.MpPourerAxis.IsHomed);
			gAxes.Timers.HomeTimer[0].PT:=REAL_TO_TIME(gAxes.TimersPar.HomeDelayTime*1000);
			gAxes.Timers.HomeTimer[0]();

			IF gAxes.Timers.HomeTimer[0].Q THEN
				gAxes.Timers.HomeTimer[0].IN:=FALSE;
				gAxes.Timers.HomeTimer[0]();
				//zbyt dlugie bazowanie osi MpCartAxis alarm
				gAxes.State.Auto:=STATE_ERROR_AXES;
			END_IF;

			IF EDGEPOS(gAxes.Ctrl.MpPourerAxis.IsHomed) THEN
				gAxes.Ctrl.MpPourerAxis.Home:=FALSE;
				gAxes.State.Manual:=STATE_WAIT_FOR_CMD_MANUAL;
				gAxes.Timers.HomeTimer[0].IN:=FALSE;
				gAxes.Timers.HomeTimer[0]();
			END_IF;
	END_CASE;

	(* Aktualizacja pozycji zmiennych wykorzystywanych w scene viewer *)
	MachineAxesPosition.Tasma:=gAxes.Ctrl.MpTransporterAxis.Position;
	MachineAxesPosition.Wozek:=gAxes.Ctrl.MpCartAxis.Position;
	MachineAxesPosition.Nalewak:=gAxes.Ctrl.MpPourerAxis.Position;;
	AdrAxesPositions:=ADR(MachineAxesPosition);

	gAxes.Ctrl.MpTransporterAxis();
	gAxes.Ctrl.MpCartAxis();
	gAxes.Ctrl.MpPourerAxis();
END_PROGRAM

PROGRAM _EXIT
	(* Insert code here *)
	gAxes.Ctrl.MpTransporterAxis.Power:=FALSE;
	gAxes.Ctrl.MpTransporterAxis.Enable:=FALSE;
	gAxes.Ctrl.MpTransporterAxis();

	gAxes.Ctrl.MpCartAxis.Power:=FALSE;
	gAxes.Ctrl.MpCartAxis.Enable:=FALSE;
	gAxes.Ctrl.MpCartAxis();

	gAxes.Ctrl.MpPourerAxis.Power:=FALSE;
	gAxes.Ctrl.MpPourerAxis.Enable:=FALSE;
	gAxes.Ctrl.MpPourerAxis();

END_PROGRAM
```

### Program Logical/Software/Code/MachineControl/MachineCtrl

#### Types.typ
```iecst
TYPE
	MachineStateType :
		(
		STATE_INIT_MACHINE := 0,
		STATE_WAIT_FOR_CMD_MACHINE := 1,
		STATE_START_MACHINE:=2,
		STATE_STOP_MACHINE:=3,
		STATE_MANUAL_MACHINE := 4,
		STATE_AUTO_MACHINE := 5,
		STATE_ESTOP_MACHINE:=6,
		STATE_ERROR_MACHINE :=7,
		STATE_HOME_TRANSPORTER_MACHINE :=8,
		STATE_HOME_CART_MACHINE := 9,
		STATE_HOME_POURER_MACHINE := 10,
		STATE_UPDATE_SPEED_MACHINE :=11,
		STATE_LOGOUT_MACHINE:=12,
		STATE_LOGIN_MACHINE:=13
	);

	StatesType : 	STRUCT
		MachineState : MachineStateType;
	END_STRUCT;

	CmdType : 	STRUCT
		MachineCmd : MachineCmdType;
	END_STRUCT;

	MachineCmdType : STRUCT
		Start : BOOL;
		Stop : BOOL;
		EStop : BOOL;
		HomeTransporter : BOOL;
		HomeCart : BOOL;
		HomePourer : BOOL;
		AutoCtrl : BOOL;
		ManualCtrl : BOOL;
		UpdateSpeed : BOOL;
		LogOut : BOOL;
		ErrorReset : BOOL;
	END_STRUCT;

	GUIType : STRUCT
		uiShowLayer : ARRAY[0..5] OF INT;
		uiShowPage : INT;
		uiCurrentPage : INT;
		uiCounterBottle : INT;
		uiConfirm : BOOL;
		uiRefuse : BOOL;
		uiAlarmStatus : BOOL;
	END_STRUCT;

	MachineCtrlType : 	STRUCT
		Timer : TON;
		Status : STRING;
		States : StatesType;
		Cmd : CmdType;
		GUI : GUIType;
	END_STRUCT;

END_TYPE
```

#### Variables.var
```iecst
VAR
	Machine :  MachineCtrlType;
END_VAR
```

#### Main.st
```iecst
PROGRAM _INIT
	(* Insert code here *)
	Machine.States.MachineState:=STATE_INIT_MACHINE;
	(* Hide all layer *)
	FOR Machine.GUI.uiShowPage:=0 TO 5 DO
		Machine.GUI.uiShowLayer[Machine.GUI.uiShowPage]:=1;
	END_FOR;

	Machine.GUI.uiShowPage:=0;
	Machine.Status:='LOGIN';
END_PROGRAM

PROGRAM _CYCLIC
	Machine.GUI.uiCounterBottle:=UDINT_TO_INT(cntButelki); //przekazanie do gui liczby nalanych butelek

	(* Warunek przejścia do stanu error | AND jest po to aby nie wchodzić tam za każdym razem i nie wyśiwetlać message boxa *)
	IF (gAxes.State.Auto=STATE_ERROR_AXES OR gCamSequencer.State=STATE_ERROR_SEQUENCER) AND (Machine.States.MachineState <> STATE_ERROR_MACHINE)THEN
		Machine.GUI.uiShowLayer[5]:=0; //message box
	  	Machine.States.MachineState:=STATE_ERROR_MACHINE;
	END_IF;

	CASE Machine.States.MachineState OF
		STATE_INIT_MACHINE:
			(* Jeśli ktoś się zaloguje  przejdź do odpowiedniej strony, która umożliwa bazowanie *)
			IF gCurrentUser <> 0 THEN
				IF Machine.GUI.uiCurrentPage=0 THEN
					Machine.Status:='INITIAL';
	  				Machine.GUI.uiShowPage:=1;
				END_IF;

				IF gAxes.State.Auto=STATE_HOME_AXES THEN
					Machine.Status:='HOMMING';
				END_IF;

				(* Jeśli osie zostały poprawnie zbazowane przejdź do main page *)
				IF gAxes.Ctrl.MpTransporterAxis.IsHomed AND gAxes.Ctrl.MpCartAxis.IsHomed AND gAxes.Ctrl.MpPourerAxis.IsHomed THEN
					Machine.GUI.uiShowPage:=2; //main page
					Machine.GUI.uiShowLayer[0]:=0;
					Machine.States.MachineState:=STATE_WAIT_FOR_CMD_MACHINE;
					Machine.Status:='WAITING';
				END_IF;
			END_IF
		STATE_WAIT_FOR_CMD_MACHINE:
			IF EDGEPOS(Machine.Cmd.MachineCmd.Start) THEN
				Machine.Cmd.MachineCmd.Start:=FALSE;
				Machine.States.MachineState:=STATE_START_MACHINE;
				//odpowiedni layer, powinien bych chyba ten co w init
			END_IF;
			IF EDGEPOS(Machine.Cmd.MachineCmd.Stop) THEN
				//stop layer -> pokazuja sie przyciski od home kazdej osi
				Machine.Cmd.MachineCmd.Stop:=FALSE;
				Machine.States.MachineState:=STATE_STOP_MACHINE;
			END_IF;
			IF EDGEPOS(Machine.Cmd.MachineCmd.ManualCtrl) THEN
				Machine.Cmd.MachineCmd.ManualCtrl:=FALSE;
				Machine.States.MachineState:=STATE_MANUAL_MACHINE;
			END_IF
			IF EDGEPOS(Machine.Cmd.MachineCmd.AutoCtrl) THEN
				Machine.Cmd.MachineCmd.AutoCtrl:=FALSE;
				Machine.States.MachineState:=STATE_AUTO_MACHINE;
			END_IF
			IF EDGEPOS(Machine.Cmd.MachineCmd.EStop) THEN
				Machine.Cmd.MachineCmd.EStop:=FALSE;
				Machine.States.MachineState:=STATE_ESTOP_MACHINE;
			END_IF
			IF EDGEPOS(Machine.Cmd.MachineCmd.HomeTransporter) THEN
				Machine.Cmd.MachineCmd.HomeTransporter:=FALSE;
				Machine.States.MachineState:=STATE_HOME_TRANSPORTER_MACHINE;
			END_IF
			IF EDGEPOS(Machine.Cmd.MachineCmd.HomeCart) THEN
				Machine.Cmd.MachineCmd.HomeCart:=FALSE;
				Machine.States.MachineState:=STATE_HOME_CART_MACHINE;
			END_IF
			IF EDGEPOS(Machine.Cmd.MachineCmd.HomePourer) THEN
				Machine.Cmd.MachineCmd.HomePourer:=FALSE;
				Machine.States.MachineState:=STATE_HOME_POURER_MACHINE;
			END_IF
			IF EDGEPOS(Machine.Cmd.MachineCmd.LogOut) THEN
				Machine.Cmd.MachineCmd.LogOut:=FALSE;
				Machine.States.MachineState:=STATE_LOGOUT_MACHINE;
			END_IF
			IF EDGEPOS(Machine.Cmd.MachineCmd.UpdateSpeed) THEN
				Machine.Cmd.MachineCmd.UpdateSpeed:=FALSE;
				Machine.States.MachineState:=STATE_UPDATE_SPEED_MACHINE;
			END_IF
			IF EDGEPOS(Machine.Cmd.MachineCmd.ErrorReset) THEN
				Machine.Cmd.MachineCmd.ErrorReset:=FALSE;
			END_IF

		STATE_START_MACHINE:
			(* Sprawdzamy czy od uruchomienia maszyny została zładowana jakakolwiek receptura *)
			IF gRecipeLoaded THEN
				(* Jeżeli poniższe inputy ustawione sa na true tzn że nalewaki, wozek są na miejscu -> można zaczynać
					Jeśli nie przechodzimy do trybu, który umieścni nalewaki i wózek na odpowiedniej pozycji
					Zabezpieczenie przed przejściem z manual do automat oraz z error do autmat*)
				IF gCamSequencer.Ctrl.MpAxisCamSequencer_0.StartSequence=TRUE AND gCamSequencer.Ctrl.MpAxisCamSequencer_1.StartSequence=TRUE THEN
					Machine.Status:='AUTOWORKING';
					gAxes.Cmd.Auto.MoveVelocity:=TRUE;
					Machine.States.MachineState:=STATE_WAIT_FOR_CMD_MACHINE;
				ELSE
					Machine.Status:='PREPARING';
					Machine.States.MachineState:=STATE_AUTO_MACHINE;
				END_IF;
			ELSE
				//wyświetlenie message boxa, że nie wczytano żadnej recipe
				Machine.GUI.uiShowLayer[2]:=0;
				Machine.States.MachineState:=STATE_WAIT_FOR_CMD_MACHINE;
			END_IF;
		STATE_STOP_MACHINE:
			Machine.Status:='STOPPED';
			gAxes.Ctrl.MpTransporterAxis.MoveVelocity:=FALSE;
			Machine.States.MachineState:=STATE_WAIT_FOR_CMD_MACHINE;
		STATE_MANUAL_MACHINE:
			//jeśli maszyna w ruchu nie przejdziesz do manual mode
			IF gAxes.Ctrl.MpTransporterAxis.MoveActive THEN
				Machine.States.MachineState:=STATE_WAIT_FOR_CMD_MACHINE;
				Machine.GUI.uiShowLayer[1]:=0; //message box
			ELSE
				Machine.Status:='MANUAL';
				Machine.GUI.uiShowPage:=6; //pokazanie strony manualnej
				gCamSequencer.Ctrl.MpAxisCamSequencer_0.StartSequence:=FALSE;
				gCamSequencer.Ctrl.MpAxisCamSequencer_1.StartSequence:=FALSE;
				gCamSequencer.Ctrl.MpAxisCamSequencer_0.EndSequence:=TRUE;
				gCamSequencer.Ctrl.MpAxisCamSequencer_1.EndSequence:=TRUE;
				Machine.States.MachineState:=STATE_WAIT_FOR_CMD_MACHINE;
			END_IF;
		STATE_AUTO_MACHINE:

			IF gAxes.Ctrl.MpTransporterAxis.MoveActive OR gAxes.Ctrl.MpTransporterAxis.MoveActive OR gAxes.Ctrl.MpPourerAxis.MoveActive THEN
				//zabezpieczenie ze jesli jest w ruchu to nie mozna z manual do auto
			ELSE
				(* Jeśli nalewaki nie są w pozycji 0 -> moveabsolute *)
				IF gAxes.Ctrl.MpPourerAxis.Position <> 0 THEN
					gAxes.Ctrl.MpPourerAxis.MoveAbsolute:=TRUE;
				ELSE
					gAxes.Ctrl.MpPourerAxis.MoveAbsolute:=FALSE;
				END_IF

				(* Powrót wózka do 0 gdy nalewaki są w 0 *)
				IF gAxes.Ctrl.MpCartAxis.Position <> 0 AND gAxes.Ctrl.MpPourerAxis.Position=0 THEN
					gAxes.Ctrl.MpCartAxis.MoveAbsolute:=TRUE;
				ELSE
					gAxes.Ctrl.MpCartAxis.MoveAbsolute:=FALSE;
				END_IF

				(* Kiedy wózek i nalewaki są na odpowiednim miejscu, można przygotować cam seq
					Przejść do znowu do poprzedniego stanu i uruchomić maszyne*)
				IF gAxes.Ctrl.MpPourerAxis.Position=0 AND gAxes.Ctrl.MpCartAxis.Position=0 THEN
					gCamSequencer.Ctrl.MpAxisCamSequencer_0.EndSequence:=FALSE;
					gCamSequencer.Ctrl.MpAxisCamSequencer_1.EndSequence:=FALSE;
					gCamSequencer.Ctrl.MpAxisCamSequencer_0.StartSequence:=TRUE;
					gCamSequencer.Ctrl.MpAxisCamSequencer_1.StartSequence:=TRUE;
					Machine.States.MachineState:=STATE_START_MACHINE;
				END_IF
			END_IF;
		STATE_HOME_TRANSPORTER_MACHINE:
			(* Jesli oś się porusza nie wyukona sie bazowanie *)
			IF gAxes.Ctrl.MpTransporterAxis.MoveActive THEN
				Machine.States.MachineState:=STATE_WAIT_FOR_CMD_MACHINE;
			ELSE
				Machine.Status:='MANUAL HOMMING';
				gAxes.Cmd.Manual.TransporterHomming;
				IF gAxes.Ctrl.MpTransporterAxis.IsHomed THEN
					Machine.States.MachineState:=STATE_WAIT_FOR_CMD_MACHINE;
					Machine.Status:='MANUAL';
				END_IF;
			END_IF;
		STATE_HOME_CART_MACHINE:
			(* Jesli oś się porusza nie wyukona sie bazowanie *)
			IF gAxes.Ctrl.MpPourerAxis.MoveActive THEN
				Machine.States.MachineState:=STATE_WAIT_FOR_CMD_MACHINE;
			ELSE
				Machine.Status:='MANUAL HOMMING';
				gAxes.Cmd.Manual.CartHomming:=TRUE;
				IF gAxes.Ctrl.MpCartAxis.IsHomed THEN
					Machine.States.MachineState:=STATE_WAIT_FOR_CMD_MACHINE;
					Machine.Status:='MANUAL';
				END_IF;
			END_IF;
		STATE_HOME_POURER_MACHINE:
			(* Jesli oś się porusza nie wyukona sie bazowanie *)
			IF gAxes.Ctrl.MpCartAxis.MoveActive THEN
				Machine.States.MachineState:=STATE_WAIT_FOR_CMD_MACHINE;
			ELSE
				Machine.Status:='MANUAL HOMMING';
				gAxes.Cmd.Manual.PourerHomming:=TRUE;
				IF gAxes.Ctrl.MpPourerAxis.IsHomed THEN
					Machine.States.MachineState:=STATE_WAIT_FOR_CMD_MACHINE;
					Machine.Status:='MANUAL';
				END_IF;
			END_IF;
		STATE_LOGOUT_MACHINE:
			(* Zabezpieczenie uniemożliwiające wylogowanie kiedy maszyna w ruchu  *)
			IF gAxes.Ctrl.MpTransporterAxis.MoveActive THEN
				Machine.States.MachineState:=STATE_WAIT_FOR_CMD_MACHINE;
				Machine.GUI.uiShowLayer[3]:=0;//message box
			ELSE
				Machine.GUI.uiShowLayer[4]:=0;//message box
				IF Machine.GUI.uiConfirm THEN //potwierdzenie wylogowanaia
					gLogOutUser:=TRUE;
					(* Jeśli nikt nie jest zalogowany tzn ze został wylogowany -> pokaż stronę z logowaniem *)
					IF gCurrentUser=0 THEN
						Machine.Status:='LOGOUT';
						Machine.GUI.uiShowLayer[4]:=1;
						Machine.States.MachineState:=STATE_LOGIN_MACHINE;
						Machine.GUI.uiShowPage:=0;
						gLogOutUser:=FALSE;
						Machine.GUI.uiConfirm:=0;
					END_IF;
				(* odrzucenie logout *)
				ELSIF Machine.GUI.uiRefuse THEN
					Machine.GUI.uiShowLayer[4]:=1;
					Machine.GUI.uiRefuse:=0;
					Machine.States.MachineState:=STATE_WAIT_FOR_CMD_MACHINE;
				END_IF;
			END_IF;
		STATE_LOGIN_MACHINE:
			(* oczekiwanie na zalogowanie i przejście do main page *)
			IF gCurrentUser>0 THEN
				Machine.GUI.uiShowPage:=2;
				Machine.States.MachineState:=STATE_WAIT_FOR_CMD_MACHINE;
			END_IF;

		STATE_UPDATE_SPEED_MACHINE:
			(* aktualizacja prędkości maszyny z poziomu gui, nie recipe *)
			gAxes.Ctrl.MpTransporterAxisPar.Velocity:=uiBottlePerMinute;
			uiBottlePerHour:=uiBottlePerMinute;
			gRecipeValues[2].Velocity:=gAxes.Ctrl.MpTransporterAxisPar.Velocity;
	        gAxes.Cmd.Auto.Update:=TRUE;
			Machine.States.MachineState:=STATE_WAIT_FOR_CMD_MACHINE;
		STATE_ERROR_MACHINE:
			(* Jeśli błąd to kończymy sekwencje  *)
			gCamSequencer.Ctrl.MpAxisCamSequencer_0.StartSequence:=FALSE;
			gCamSequencer.Ctrl.MpAxisCamSequencer_1.StartSequence:=FALSE;
			gCamSequencer.Ctrl.MpAxisCamSequencer_0.EndSequence:=TRUE;
			gCamSequencer.Ctrl.MpAxisCamSequencer_1.EndSequence:=TRUE;

			Machine.Timer.IN:=NOT(Machine.Timer.Q);
			Machine.Timer.PT:=T#300ms;
			Machine.Timer();

			Machine.GUI.uiAlarmStatus:=Machine.GUI.uiAlarmStatus XOR Machine.Timer.Q;

			IF EDGEPOS(Machine.Cmd.MachineCmd.ErrorReset)THEN
				Machine.Cmd.MachineCmd.ErrorReset:=FALSE;
				gAxes.Cmd.Auto.ErrorReset:=TRUE;
				gCamSequencer.Cmd.ErrorReset:=TRUE;
			END_IF;

			(* Okienko message box jeśli confirm przenosi na alarmy jeśli refuse znika *)
			IF EDGEPOS(Machine.GUI.uiConfirm) THEN
				Machine.GUI.uiConfirm:=0;
				Machine.GUI.uiShowLayer[5]:=1;
				Machine.GUI.uiShowPage:=3;
			ELSIF EDGEPOS(Machine.GUI.uiRefuse) THEN
				Machine.GUI.uiShowLayer[5]:=1;
				Machine.GUI.uiRefuse:=0;
			END_IF

			(* jeśli nie ma błędów przejdz do odpowiedniego stanu *)
			IF gAxes.State.Auto<>STATE_ERROR_AXES AND gCamSequencer.State<>STATE_ERROR_SEQUENCER THEN
				Machine.GUI.uiAlarmStatus:=0;
				Machine.Timer.IN:=FALSE;
				Machine.Timer();
				Machine.States.MachineState:=STATE_WAIT_FOR_CMD_MACHINE;
			END_IF;
	END_CASE;
END_PROGRAM

PROGRAM _EXIT
	(* Insert code here *)

END_PROGRAM
```

### RecipeCtrlGlobal.typ
```iecst
TYPE
	gRecipeValuesType : 	STRUCT
		Velocity : REAL;
		MasterFactor : DINT;
		SlaveFactor : DINT;
		Height : REAL;
		Volume : REAL;
	END_STRUCT;
END_TYPE
```

### RecipeCtrlGlobal.var
```iecst
VAR
	gRecipeValues : ARRAY[2..4] OF gRecipeValuesType;
	gRecipeLoaded : BOOL;
	uiBottlePerMinute : REAL;
	uiBottlePerHour : REAL;
	uiRecipeBottlePerMinute : REAL;
	uiRecipeBottlePerHour : REAL;
END_VAR
```

### Program Logical/Software/Code/RecipeControl/RecipeCtrl

#### Types.typ
```iecst
TYPE
	RecipeCtrlType : STRUCT
		RecipeXml : MpRecipeXml;
		RecipeRegPar : MpRecipeRegPar;

		RecipeUI : MpRecipeUI;
		RecipeUISetup : MpRecipeUISetupType;
		RecipeUIConnect : MpRecipeUIConnectType;

		RecipeData : RecipeDataType;

		FileManagerUI : MpFileManagerUI;
		FileManagerSetup : MpFileManagerUISetupType;
		FileManagerUIConnect : MpFileManagerUIConnectType;

		State : RecipeState;
		Cmd : RecipeCmdType;
		RecipeEdit : RecipeEditType;
		RecipeDefaultValues : ARRAY[2..4] OF RecipeDefaultValuesType;
	END_STRUCT;

	RecipeDefaultValuesType : STRUCT
		Velocity : REAL;
		Height : REAL;
		Volume : REAL;
		MasterFactor : DINT;
		SlaveFactor : DINT;
	END_STRUCT;

	RecipeDataType : STRUCT
		DeviceName : STRING[20] := 'RecipeFile';
		FileName : STRING[20]:='MyRecipe';
	END_STRUCT;

	RecipeCmdType : STRUCT
		Load : BOOL;
		Save : BOOL;
		Edit : BOOL;
		SaveEdit : BOOL;
	END_STRUCT;

	RecipeEditType : STRUCT
		Height1 : REAL;
		Height2 : REAL;
		Height3 : REAL;
		Volume1 : REAL;
		Volume2 : REAL;
		BottlePerMinute : REAL;
		Factor : REAL;
		Distance1 : REAL;
		Distance2 : REAL;
		Distance3 : REAL;
		Name : STRING;
	END_STRUCT;

	RecipeState :
		(
		STATE_LOAD_RECIPE := 2,
		STATE_SAVE_RECIPE := 1,
		STATE_EDIT_RECIPE := 5,
		STATE_INIT_RECIPE :=4,
		STATE_WAIT_RECIPE :=0
	);

END_TYPE
```

#### Main.st
```iecst
PROGRAM _INIT
	(* Insert code here *)
	Recipe.RecipeXml.Enable:=TRUE;
	Recipe.RecipeUI.Enable:=TRUE;
	Recipe.RecipeRegPar.Enable:=TRUE;
	Recipe.FileManagerUI.Enable:=TRUE;

	Recipe.RecipeDefaultValues[2].Velocity:=100;
	Recipe.RecipeDefaultValues[2].Height:=90;
	Recipe.RecipeDefaultValues[2].Volume:=400;
	Recipe.RecipeDefaultValues[2].MasterFactor:=215*100;
	Recipe.RecipeDefaultValues[2].SlaveFactor:=-90*100;

	Recipe.RecipeDefaultValues[3].Velocity:=100;
	Recipe.RecipeDefaultValues[3].Height:=65;
	Recipe.RecipeDefaultValues[3].Volume:=100;
	Recipe.RecipeDefaultValues[3].MasterFactor:=54*100;
	Recipe.RecipeDefaultValues[3].SlaveFactor:=-65*100;

	Recipe.RecipeDefaultValues[4].Velocity:=100;
	Recipe.RecipeDefaultValues[4].Height:=60;
	Recipe.RecipeDefaultValues[4].Volume:=0;
	Recipe.RecipeDefaultValues[4].MasterFactor:=22*100;
	Recipe.RecipeDefaultValues[4].SlaveFactor:=-60*100;

	(* DEFAULT FALUES FOR RECIPE *)
	gRecipeValues[2].Velocity:=Recipe.RecipeDefaultValues[2].Velocity;
	gRecipeValues[2].Height:=Recipe.RecipeDefaultValues[2].Height;
	gRecipeValues[2].Volume:=Recipe.RecipeDefaultValues[2].Volume;
	gRecipeValues[2].MasterFactor:=Recipe.RecipeDefaultValues[2].MasterFactor;
	gRecipeValues[2].SlaveFactor:=Recipe.RecipeDefaultValues[2].SlaveFactor;

	gRecipeValues[3].Velocity:=Recipe.RecipeDefaultValues[3].Velocity;
	gRecipeValues[3].Height:=Recipe.RecipeDefaultValues[3].Height;
	gRecipeValues[3].Volume:=Recipe.RecipeDefaultValues[3].Volume;
	gRecipeValues[3].MasterFactor:=Recipe.RecipeDefaultValues[3].MasterFactor;
	gRecipeValues[3].SlaveFactor:=Recipe.RecipeDefaultValues[3].SlaveFactor;

	gRecipeValues[4].Velocity:=Recipe.RecipeDefaultValues[4].Velocity;
	gRecipeValues[4].Height:=Recipe.RecipeDefaultValues[4].Height;
	gRecipeValues[4].MasterFactor:=Recipe.RecipeDefaultValues[4].MasterFactor;
	gRecipeValues[4].SlaveFactor:=Recipe.RecipeDefaultValues[4].SlaveFactor;

	Recipe.State:=STATE_INIT_RECIPE;
	gRecipeLoaded:=TRUE;
END_PROGRAM

PROGRAM _CYCLIC
	(* Insert code here *)
	Recipe.RecipeXml.MpLink:=ADR(gRecipeXml);
	Recipe.RecipeXml.DeviceName:=ADR(Recipe.RecipeData.DeviceName);
	Recipe.RecipeXml.FileName:=ADR('DefaultRecipe');

	Recipe.RecipeUI.MpLink:=ADR(gRecipeXml);
	Recipe.RecipeUI.UIConnect:=ADR(Recipe.RecipeUIConnect);

	Recipe.RecipeUISetup.Confirmation.RecipeLoad:=TRUE;
	Recipe.RecipeUISetup.Confirmation.RecipeDelete:=TRUE;
	Recipe.RecipeUISetup.Confirmation.RecipeSave:=TRUE;
	Recipe.RecipeUISetup.Confirmation.RecipeCreate:=TRUE;
	Recipe.RecipeUISetup.Confirmation.RecipeRename:=TRUE;
	Recipe.RecipeUI.UISetup:=Recipe.RecipeUISetup;

	Recipe.RecipeRegPar.MpLink:=ADR(gRecipeXml);
	Recipe.RecipeRegPar.PVName:=ADR('gRecipeValues');

	Recipe.FileManagerUI.MpLink:=ADR(gFileManagerUI);
	Recipe.FileManagerUI.UIConnect:=ADR(Recipe.FileManagerUIConnect);
	Recipe.FileManagerUI.UISetup:=Recipe.FileManagerSetup;

	Recipe.FileManagerUIConnect.DeviceList.DeviceNames[0]:=Recipe.RecipeData.DeviceName;

	Recipe.RecipeEdit.Name:=Recipe.RecipeUIConnect.Recipe.List.Names[Recipe.RecipeUIConnect.Recipe.List.SelectedIndex];

	(* Maszyna stanów kontrolująca zapisywanie i wczytywanie z recipe do struktury  *)
	CASE Recipe.State OF
		STATE_INIT_RECIPE:
			(* Stan w którym zapisujemy domyślną receptruę *)
			Recipe.RecipeXml.Save:=TRUE;
			IF Recipe.RecipeXml.CommandDone THEN
				Recipe.RecipeXml.Save:=FALSE;
				Recipe.State:=STATE_WAIT_RECIPE;
			END_IF;

		STATE_WAIT_RECIPE:
			(* Jesli receptura jest wczytywana, przejdz do odpowiedniego stanu  *)
			IF Recipe.RecipeUIConnect.Status=mpRECIPE_UI_STATUS_LOAD THEN
				Recipe.State:=STATE_LOAD_RECIPE;
			(* Jeśli wyskoczył message box proszący o potwierdzenie zapisu struktury do recipe, przejdz do odpowiedniego stanu  *)
//			ELSIF Recipe.RecipeUIConnect.MessageBox.Type=mpRECIPE_UI_MSG_CONFIRM_SAVE THEN
//				Recipe.State:=STATE_SAVE_RECIPE;
			ELSIF EDGEPOS(Recipe.Cmd.Edit) THEN
				Recipe.Cmd.Edit:=FALSE;
				Recipe.State:=STATE_EDIT_RECIPE;
			END_IF;
		STATE_LOAD_RECIPE:
			(* Jesli bloczek oczekuje na cmd tzn że zostało wczytanie do struktury i można zaimplementować zmiany ze struktury do camseq *)
			IF Recipe.RecipeUIConnect.Status=mpRECIPE_UI_STATUS_IDLE THEN
				gRecipeLoaded:=TRUE; //flaga informująca że jakakolwiek receptura została waczytana

				(* Aktualizacja zmiennych z GUI *)
				uiRecipeBottlePerMinute := gRecipeValues[2].Velocity;
				uiRecipeBottlePerHour := gRecipeValues[2].Velocity;
				uiBottlePerHour:=gRecipeValues[2].Velocity;
				uiBottlePerMinute:=gRecipeValues[2].Velocity;

				(* Aktualizacja parametrów sequencera *)
				gAxes.Ctrl.MpTransporterAxisPar.Velocity:=gRecipeValues[2].Velocity;
				gCamSequencer.Ctrl.MpAxisCamSequencerPar_1.Configuration.State[2].MasterFactor:=gRecipeValues[2].MasterFactor;
				gCamSequencer.Ctrl.MpAxisCamSequencerPar_1.Configuration.State[2].SlaveFactor:=gRecipeValues[2].SlaveFactor;

				gCamSequencer.Ctrl.MpAxisCamSequencerPar_1.Configuration.State[3].MasterFactor:=gRecipeValues[3].MasterFactor;
				gCamSequencer.Ctrl.MpAxisCamSequencerPar_1.Configuration.State[3].SlaveFactor:=gRecipeValues[3].SlaveFactor;

				gCamSequencer.Ctrl.MpAxisCamSequencerPar_1.Configuration.State[4].MasterFactor:=gRecipeValues[4].MasterFactor;
				gCamSequencer.Ctrl.MpAxisCamSequencerPar_1.Configuration.State[4].SlaveFactor:=gRecipeValues[4].SlaveFactor;

				(* Update dokonanych zmian -> Update musi dokonać się w odpowiednim state aby nie popsuć pracy  *)
				IF gCamSequencer.Ctrl.MpAxisCamSequencer_0.StartSequence=TRUE AND gCamSequencer.Ctrl.MpAxisCamSequencer_0.ActualStateIndex=2 THEN
					gCamSequencer.Ctrl.MpAxisCamSequencer_1.Update:=TRUE;
					gAxes.Cmd.Auto.Update:=TRUE;
					Recipe.State:=STATE_WAIT_RECIPE;
				ELSIF gCamSequencer.Ctrl.MpAxisCamSequencer_0.StartSequence=FALSE THEN
					gCamSequencer.Ctrl.MpAxisCamSequencer_1.Update:=TRUE;
					gAxes.Cmd.Auto.Update:=TRUE;
					Recipe.State:=STATE_WAIT_RECIPE;
				END_IF
			END_IF;

		STATE_SAVE_RECIPE:
			(* Zapisanie aktualnych parametrów sequencera do struktury -> aktualizacja tylko wtedy gdy wyskoczy message box *)
			gRecipeValues[2].Velocity:=gAxes.Ctrl.MpTransporterAxisPar.Velocity;
			gRecipeValues[2].MasterFactor:=gCamSequencer.Ctrl.MpAxisCamSequencerPar_1.Configuration.State[1].MasterFactor;
			gRecipeValues[2].SlaveFactor:=gCamSequencer.Ctrl.MpAxisCamSequencerPar_1.Configuration.State[1].SlaveFactor;

			gRecipeValues[3].Velocity:=gAxes.Ctrl.MpTransporterAxisPar.Velocity;
			gRecipeValues[3].MasterFactor:=gCamSequencer.Ctrl.MpAxisCamSequencerPar_1.Configuration.State[2].MasterFactor;
			gRecipeValues[3].SlaveFactor:=gCamSequencer.Ctrl.MpAxisCamSequencerPar_1.Configuration.State[2].SlaveFactor;

			gRecipeValues[4].Velocity:=gAxes.Ctrl.MpTransporterAxisPar.Velocity;
			gRecipeValues[4].MasterFactor:=gCamSequencer.Ctrl.MpAxisCamSequencerPar_1.Configuration.State[3].MasterFactor;
			gRecipeValues[4].SlaveFactor:=gCamSequencer.Ctrl.MpAxisCamSequencerPar_1.Configuration.State[3].SlaveFactor;

			Recipe.State:=STATE_WAIT_RECIPE;

		STATE_EDIT_RECIPE:
			Recipe.RecipeEdit.Height3:=215-(Recipe.RecipeEdit.Height1 + Recipe.RecipeEdit.Height2 );
			Recipe.RecipeEdit.Distance3:=Recipe.RecipeEdit.Height3/2.75; (* Współczynnik wzięty ze stosunku przebytej drogi do odleglosci na ktora zjezdza nalewak *)
			Recipe.RecipeEdit.Factor:=(290-Recipe.RecipeEdit.Distance3)/(Recipe.RecipeEdit.Volume1+Recipe.RecipeEdit.Volume2);
			Recipe.RecipeEdit.Distance1:=Recipe.RecipeEdit.Factor*Recipe.RecipeEdit.Volume1;
			Recipe.RecipeEdit.Distance2:=Recipe.RecipeEdit.Factor*Recipe.RecipeEdit.Volume2;

			gRecipeValues[2].Velocity:=Recipe.RecipeEdit.BottlePerMinute;
			gRecipeValues[2].MasterFactor:=REAL_TO_DINT(Recipe.RecipeEdit.Distance1)*100;
			gRecipeValues[2].SlaveFactor:=REAL_TO_DINT(-Recipe.RecipeEdit.Height1)*100;
			gRecipeValues[2].Height:=Recipe.RecipeEdit.Height1;
			gRecipeValues[2].Volume:=Recipe.RecipeEdit.Volume1;

			gRecipeValues[3].Velocity:=Recipe.RecipeEdit.BottlePerMinute;
			gRecipeValues[3].MasterFactor:=REAL_TO_DINT(Recipe.RecipeEdit.Distance2)*100;
			gRecipeValues[3].SlaveFactor:=REAL_TO_DINT(-Recipe.RecipeEdit.Height2)*100;
			gRecipeValues[3].Height:=Recipe.RecipeEdit.Height2;
			gRecipeValues[3].Volume:=Recipe.RecipeEdit.Volume2;

			gRecipeValues[4].Velocity:=Recipe.RecipeEdit.BottlePerMinute;
			gRecipeValues[4].MasterFactor:=REAL_TO_DINT(Recipe.RecipeEdit.Distance3)*100;
			gRecipeValues[4].SlaveFactor:=REAL_TO_DINT(-Recipe.RecipeEdit.Height3)*100;

			Recipe.RecipeUIConnect.Recipe.Save:=TRUE;
			Recipe.RecipeUIConnect.Recipe.Refresh:=FALSE;
			IF Recipe.RecipeUIConnect.MessageBox.LayerStatus=0 THEN
				Recipe.RecipeUIConnect.Recipe.Save:=FALSE;
				Recipe.State:=STATE_WAIT_RECIPE;
			END_IF;

			(* Do zrobienia zapamietanie indexu zaznaczonego poniewaz po zapisie wybrany index wraca na 0 *)
			(* Tez popup *) (* albo dorobić zeby wychodzuło i tyle i popup ze nalezy wczytac  *)
//			Recipe.RecipeXml.FileName:=ADR(Recipe.RecipeUIConnect.Recipe.List.Names[Recipe.RecipeUIConnect.Recipe.List.SelectedIndex]);
//			Recipe.RecipeXml.Save:=TRUE;
//			IF Recipe.RecipeXml.CommandDone THEN
//				Recipe.RecipeXml.Save:=FALSE;
//				Recipe.State:=STATE_WAIT_RECIPE;
//			END_IF;
	END_CASE;

	Recipe.RecipeXml();
	Recipe.RecipeRegPar();
	Recipe.RecipeUI();
	Recipe.FileManagerUI();
END_PROGRAM

PROGRAM _EXIT
	(* Insert code here *)

END_PROGRAM
```

### SequencerCtrlGlobal.typ
```iecst
TYPE
	gCamSequencerStateType :
		(
		STATE_ERROR_SEQUENCER := 1,
		STATE_WORK_SEQUENCER := 0
		);
	gCamSequencerCmdType : 	STRUCT
		ErrorReset : BOOL;
	END_STRUCT;
	gCamSequencerCtrlType : 	STRUCT
		Ctrl : gCamSequencerBasicCtrlType;
		State : gCamSequencerStateType;
		Cmd : gCamSequencerCmdType;
	END_STRUCT;
	gCamSequencerBasicCtrlType : 	STRUCT
		MpAxisCamSequencer_0 : MpAxisCamSequencer;
		MpAxisCamSequencerPar_0 : MpAxisCamSequencerParType;
		MpAxisCamSequencer_1 : MpAxisCamSequencer;
		MpAxisCamSequencerPar_1 : MpAxisCamSequencerParType;
	END_STRUCT;
END_TYPE
```

### SequencerCtrlGlobal.var
```iecst
VAR
	gCamSequencer : gCamSequencerCtrlType;
END_VAR
```

### Program Logical/Software/Code/SequencerControl/SequencerCtrl

#### Variables.var
```iecst
VAR
	DoPourer : BOOL;
END_VAR

VAR CONSTANT

END_VAR
```
